    |   movel([0.162608, -1.218447, -2.664024, -0.829918, 1.570796, 1.733404],accel_mss,speed_ms,0,blend_radius_m)
    |   movel([0.161685, -1.220294, -2.663101, -0.828994, 1.570796, 1.732481],accel_mss,speed_ms,0,blend_radius_m)
    |   movel([0.160585, -1.222184, -2.662153, -0.828052, 1.570796, 1.731381],accel_mss,speed_ms,0,blend_radius_m)
    |   movel([0.163671, -1.223075, -2.661704, -0.827609, 1.570796, 1.734467],accel_mss,speed_ms,0,blend_radius_m)
    |   movel([0.165524, -1.220284, -2.663106, -0.828999, 1.570796, 1.736320],accel_mss,speed_ms,0,blend_radius_m)
    |   speed_ms = 0.005
    |   # Splitting Linear movement in 4 (instruction 1016: MoveL 952)
    |   movel([0.165524, -1.217896, -2.661930, -0.832564, 1.570796, 1.736320],accel_mss,speed_ms,0,blend_radius_m)
    |   movel([0.165524, -1.215522, -2.660749, -0.836117, 1.570796, 1.736320],accel_mss,speed_ms,0,blend_radius_m)
    |   movel([0.165524, -1.213164, -2.659566, -0.839659, 1.570796, 1.736320],accel_mss,speed_ms,0,blend_radius_m)
    |   movel([0.165524, -1.210820, -2.658378, -0.843191, 1.570796, 1.736320],accel_mss,speed_ms,0,blend_radius_m)
    |   speed_ms = 0.040
    |   # Splitting Linear movement in 8 (instruction 1018: MoveL 953)
    |   movel([0.167766, -1.211543, -2.658021, -0.842825, 1.570796, 1.738562],accel_mss,speed_ms,0,blend_radius_m)
    |   movel([0.170001, -1.212273, -2.657659, -0.842457, 1.570796, 1.740797],accel_mss,speed_ms,0,blend_radius_m)
    |   movel([0.172230, -1.213009, -2.657294, -0.842086, 1.570796, 1.743026],accel_mss,speed_ms,0,blend_radius_m)
    |   movel([0.174452, -1.213751, -2.656925, -0.841713, 1.570796, 1.745249],accel_mss,speed_ms,0,blend_radius_m)
    |   movel([0.176668, -1.214500, -2.656552, -0.841337, 1.570796, 1.747465],accel_mss,speed_ms,0,blend_radius_m)
    |   movel([0.178878, -1.215256, -2.656175, -0.840958, 1.570796, 1.749674],accel_mss,speed_ms,0,blend_radius_m)
    |   movel([0.181081, -1.216017, -2.655795, -0.840577, 1.570796, 1.751878],accel_mss,speed_ms,0,blend_radius_m)
    |   movel([0.183278, -1.216785, -2.655410, -0.840194, 1.570796, 1.754074],accel_mss,speed_ms,0,blend_radius_m)
    |   speed_ms = 0.005
    |   # Splitting Linear movement in 4 (instruction 1020: MoveL 954)
    |   movel([0.183278, -1.219124, -2.656591, -0.836674, 1.570796, 1.754074],accel_mss,speed_ms,0,blend_radius_m)
    |   movel([0.183278, -1.221477, -2.657768, -0.833145, 1.570796, 1.754074],accel_mss,speed_ms,0,blend_radius_m)
    |   movel([0.183278, -1.223844, -2.658941, -0.829604, 1.570796, 1.754074],accel_mss,speed_ms,0,blend_radius_m)
    |   movel([0.183278, -1.226226, -2.660111, -0.826052, 1.570796, 1.754074],accel_mss,speed_ms,0,blend_radius_m)
    |   speed_ms = 0.035
    |   movel([0.185050, -1.223552, -2.661464, -0.827373, 1.570796, 1.755846],accel_mss,speed_ms,0,blend_radius_m)
    |   movel([0.186685, -1.220770, -2.662863, -0.828756, 1.570796, 1.757481],accel_mss,speed_ms,0,blend_radius_m)
    |   movel([0.188167, -1.217900, -2.664296, -0.830193, 1.570796, 1.758964],accel_mss,speed_ms,0,blend_radius_m)
    |   movel([0.189493, -1.214960, -2.665755, -0.831674, 1.570796, 1.760289],accel_mss,speed_ms,0,blend_radius_m)
    |   movel([0.190642, -1.211967, -2.667230, -0.833191, 1.570796, 1.761439],accel_mss,speed_ms,0,blend_radius_m)
    |   movel([0.191604, -1.208945, -2.668710, -0.834734, 1.570796, 1.762401],accel_mss,speed_ms,0,blend_radius_m)
    |   movel([0.192368, -1.205907, -2.670187, -0.836295, 1.570796, 1.763165],accel_mss,speed_ms,0,blend_radius_m)
    |   movel([0.192919, -1.202878, -2.671649, -0.837862, 1.570796, 1.763715],accel_mss,speed_ms,0,blend_radius_m)
    |   movel([0.193243, -1.199877, -2.673088, -0.839424, 1.570796, 1.764039],accel_mss,speed_ms,0,blend_radius_m)
    |   movel([0.193330, -1.196922, -2.674495, -0.840972, 1.570796, 1.764126],accel_mss,speed_ms,0,blend_radius_m)
    |   movel([0.193159, -1.194041, -2.675858, -0.842490, 1.570796, 1.763955],accel_mss,speed_ms,0,blend_radius_m)
    |   movel([0.192720, -1.191255, -2.677167, -0.843967, 1.570796, 1.763517],accel_mss,speed_ms,0,blend_radius_m)
    |   movel([0.192000, -1.188584, -2.678414, -0.845391, 1.570796, 1.762796],accel_mss,speed_ms,0,blend_radius_m)
    |   movel([0.190984, -1.186054, -2.679588, -0.846746, 1.570796, 1.761780],accel_mss,speed_ms,0,blend_radius_m)
    |   movel([0.189658, -1.183690, -2.680680, -0.848019, 1.570796, 1.760454],accel_mss,speed_ms,0,blend_radius_m)
    |   movel([0.188006, -1.181513, -2.681679, -0.849197, 1.570796, 1.758802],accel_mss,speed_ms,0,blend_radius_m)
    |   movel([0.186034, -1.179579, -2.682563, -0.850247, 1.570796, 1.756830],accel_mss,speed_ms,0,blend_radius_m)
    |   movel([0.183805, -1.177953, -2.683303, -0.851133, 1.570796, 1.754602],accel_mss,speed_ms,0,blend_radius_m)
    |   movel([0.181340, -1.176638, -2.683899, -0.851852, 1.570796, 1.752136],accel_mss,speed_ms,0,blend_radius_m)
    |   movel([0.178653, -1.175637, -2.684352, -0.852400, 1.570796, 1.749450],accel_mss,speed_ms,0,blend_radius_m)
    |   movel([0.175765, -1.174950, -2.684662, -0.852777, 1.570796, 1.746561],accel_mss,speed_ms,0,blend_radius_m)
    |   movel([0.172695, -1.174575, -2.684831, -0.852983, 1.570796, 1.743491],accel_mss,speed_ms,0,blend_radius_m)
    |   movel([0.169469, -1.174511, -2.684860, -0.853018, 1.570796, 1.740265],accel_mss,speed_ms,0,blend_radius_m)
    |   movel([0.166102, -1.174756, -2.684749, -0.852884, 1.570796, 1.736898],accel_mss,speed_ms,0,blend_radius_m)
    |   movel([0.162621, -1.175304, -2.684502, -0.852583, 1.570796, 1.733417],accel_mss,speed_ms,0,blend_radius_m)
    |   movel([0.159044, -1.176159, -2.684116, -0.852114, 1.570796, 1.729840],accel_mss,speed_ms,0,blend_radius_m)
    |   movel([0.155393, -1.177310, -2.683594, -0.851484, 1.570796, 1.726189],accel_mss,speed_ms,0,blend_radius_m)
    |   movel([0.151692, -1.178755, -2.682938, -0.850696, 1.570796, 1.722489],accel_mss,speed_ms,0,blend_radius_m)
    |   movel([0.147964, -1.180489, -2.682147, -0.849753, 1.570796, 1.718760],accel_mss,speed_ms,0,blend_radius_m)
    |   movel([0.144226, -1.182504, -2.681225, -0.848661, 1.570796, 1.715023],accel_mss,speed_ms,0,blend_radius_m)
    |   movel([0.140507, -1.184794, -2.680171, -0.847424, 1.570796, 1.711304],accel_mss,speed_ms,0,blend_radius_m)
    |   movel([0.136826, -1.187352, -2.678987, -0.846050, 1.570796, 1.707622],accel_mss,speed_ms,0,blend_radius_m)
    |   movel([0.133191, -1.190174, -2.677673, -0.844542, 1.570796, 1.703987],accel_mss,speed_ms,0,blend_radius_m)
    |   movel([0.129733, -1.193158, -2.676274, -0.842957, 1.570796, 1.700530],accel_mss,speed_ms,0,blend_radius_m)
    |   movel([0.126470, -1.196275, -2.674802, -0.841312, 1.570796, 1.697266],accel_mss,speed_ms,0,blend_radius_m)
    |   movel([0.123412, -1.199505, -2.673266, -0.839619, 1.570796, 1.694208],accel_mss,speed_ms,0,blend_radius_m)
    |   movel([0.120568, -1.202823, -2.671675, -0.837890, 1.570796, 1.691365],accel_mss,speed_ms,0,blend_radius_m)
    |   movel([0.117952, -1.206214, -2.670038, -0.836137, 1.570796, 1.688748],accel_mss,speed_ms,0,blend_radius_m)
    |   movel([0.115566, -1.209658, -2.668362, -0.834369, 1.570796, 1.686363],accel_mss,speed_ms,0,blend_radius_m)
    |   movel([0.113428, -1.213130, -2.666659, -0.832601, 1.570796, 1.684225],accel_mss,speed_ms,0,blend_radius_m)
    |   movel([0.111540, -1.216616, -2.664935, -0.830838, 1.570796, 1.682336],accel_mss,speed_ms,0,blend_radius_m)
    |   movel([0.109910, -1.220098, -2.663199, -0.829092, 1.570796, 1.680707],accel_mss,speed_ms,0,blend_radius_m)
    |   movel([0.108548, -1.223555, -2.661462, -0.827371, 1.570796, 1.679344],accel_mss,speed_ms,0,blend_radius_m)
    |   movel([0.107464, -1.226975, -2.659731, -0.825683, 1.570796, 1.678260],accel_mss,speed_ms,0,blend_radius_m)
    |   movel([0.106659, -1.230338, -2.658015, -0.824036, 1.570796, 1.677455],accel_mss,speed_ms,0,blend_radius_m)
    |   movel([0.106148, -1.233627, -2.656324, -0.822437, 1.570796, 1.676944],accel_mss,speed_ms,0,blend_radius_m)
    |   movel([0.105928, -1.236831, -2.654665, -0.820893, 1.570796, 1.676724],accel_mss,speed_ms,0,blend_radius_m)
    |   movel([0.106013, -1.239934, -2.653047, -0.819408, 1.570796, 1.676809],accel_mss,speed_ms,0,blend_radius_m)
    |   movel([0.106368, -1.242656, -2.651618, -0.818114, 1.570796, 1.677165],accel_mss,speed_ms,0,blend_radius_m)
    |   movel([0.106979, -1.245156, -2.650298, -0.816935, 1.570796, 1.677775],accel_mss,speed_ms,0,blend_radius_m)
    |   movel([0.107817, -1.247439, -2.649086, -0.815864, 1.570796, 1.678614],accel_mss,speed_ms,0,blend_radius_m)
    |   movel([0.108863, -1.249512, -2.647981, -0.814897, 1.570796, 1.679659],accel_mss,speed_ms,0,blend_radius_m)
    |   movel([0.110091, -1.251379, -2.646980, -0.814030, 1.570796, 1.680887],accel_mss,speed_ms,0,blend_radius_m)
    |   movel([0.111476, -1.253047, -2.646083, -0.813259, 1.570796, 1.682272],accel_mss,speed_ms,0,blend_radius_m)
    |   movel([0.112995, -1.254520, -2.645288, -0.812581, 1.570796, 1.683792],accel_mss,speed_ms,0,blend_radius_m)
    |   movel([0.114629, -1.255802, -2.644593, -0.811993, 1.570796, 1.685426],accel_mss,speed_ms,0,blend_radius_m)
    |   movel([0.116356, -1.256897, -2.643999, -0.811493, 1.570796, 1.687152],accel_mss,speed_ms,0,blend_radius_m)
    |   movel([0.118150, -1.257811, -2.643502, -0.811076, 1.570796, 1.688947],accel_mss,speed_ms,0,blend_radius_m)
    |   movel([0.119994, -1.258543, -2.643103, -0.810743, 1.570796, 1.690791],accel_mss,speed_ms,0,blend_radius_m)
    |   movel([0.121863, -1.259101, -2.642798, -0.810490, 1.570796, 1.692659],accel_mss,speed_ms,0,blend_radius_m)
    |   movel([0.123738, -1.259483, -2.642589, -0.810316, 1.570796, 1.694534],accel_mss,speed_ms,0,blend_radius_m)
    |   movel([0.125599, -1.259692, -2.642475, -0.810222, 1.570796, 1.696395],accel_mss,speed_ms,0,blend_radius_m)
    |   movel([0.127421, -1.259733, -2.642453, -0.810203, 1.570796, 1.698217],accel_mss,speed_ms,0,blend_radius_m)
    |   movel([0.129187, -1.259604, -2.642523, -0.810261, 1.570796, 1.699983],accel_mss,speed_ms,0,blend_radius_m)
    |   movel([0.130799, -1.256111, -2.644426, -0.811852, 1.570796, 1.701596],accel_mss,speed_ms,0,blend_radius_m)
    |   movel([0.127034, -1.255651, -2.644675, -0.812062, 1.570796, 1.697831],accel_mss,speed_ms,0,blend_radius_m)
    |   movel([0.123670, -1.254813, -2.645129, -0.812447, 1.570796, 1.694467],accel_mss,speed_ms,0,blend_radius_m)
    |   movel([0.120699, -1.253624, -2.645772, -0.812993, 1.570796, 1.691495],accel_mss,speed_ms,0,blend_radius_m)
    |   movel([0.118110, -1.252108, -2.646588, -0.813693, 1.570796, 1.688906],accel_mss,speed_ms,0,blend_radius_m)
    |   movel([0.115901, -1.250284, -2.647567, -0.814538, 1.570796, 1.686697],accel_mss,speed_ms,0,blend_radius_m)
    |   movel([0.114064, -1.248180, -2.648692, -0.815517, 1.570796, 1.684861],accel_mss,speed_ms,0,blend_radius_m)
    |   movel([0.112599, -1.245812, -2.649950, -0.816626, 1.570796, 1.683395],accel_mss,speed_ms,0,blend_radius_m)
    |   movel([0.111497, -1.243210, -2.651326, -0.817853, 1.570796, 1.682294],accel_mss,speed_ms,0,blend_radius_m)
    |   movel([0.110757, -1.240392, -2.652807, -0.819190, 1.570796, 1.681553],accel_mss,speed_ms,0,blend_radius_m)
    |   movel([0.110373, -1.237384, -2.654378, -0.820627, 1.570796, 1.681169],accel_mss,speed_ms,0,blend_radius_m)
    |   movel([0.110346, -1.234208, -2.656024, -0.822156, 1.570796, 1.681143],accel_mss,speed_ms,0,blend_radius_m)
    |   movel([0.110668, -1.230893, -2.657731, -0.823765, 1.570796, 1.681464],accel_mss,speed_ms,0,blend_radius_m)
    |   movel([0.111341, -1.227459, -2.659485, -0.825445, 1.570796, 1.682137],accel_mss,speed_ms,0,blend_radius_m)
    |   movel([0.112362, -1.223936, -2.661270, -0.827183, 1.570796, 1.683158],accel_mss,speed_ms,0,blend_radius_m)
    |   movel([0.113724, -1.220347, -2.663074, -0.828967, 1.570796, 1.684520],accel_mss,speed_ms,0,blend_radius_m)
    |   movel([0.115426, -1.216725, -2.664880, -0.830783, 1.570796, 1.686223],accel_mss,speed_ms,0,blend_radius_m)
    |   movel([0.117544, -1.212934, -2.666755, -0.832700, 1.570796, 1.688341],accel_mss,speed_ms,0,blend_radius_m)
    |   movel([0.119932, -1.209242, -2.668565, -0.834582, 1.570796, 1.690729],accel_mss,speed_ms,0,blend_radius_m)
    |   movel([0.122570, -1.205662, -2.670305, -0.836421, 1.570796, 1.693366],accel_mss,speed_ms,0,blend_radius_m)
    |   movel([0.125434, -1.202220, -2.671966, -0.838204, 1.570796, 1.696231],accel_mss,speed_ms,0,blend_radius_m)
    |   movel([0.128500, -1.198935, -2.673537, -0.839916, 1.570796, 1.699296],accel_mss,speed_ms,0,blend_radius_m)
    |   movel([0.131747, -1.195825, -2.675015, -0.841549, 1.570796, 1.702544],accel_mss,speed_ms,0,blend_radius_m)
    |   movel([0.135148, -1.192915, -2.676388, -0.843086, 1.570796, 1.705945],accel_mss,speed_ms,0,blend_radius_m)
    |   movel([0.138679, -1.190222, -2.677650, -0.844517, 1.570796, 1.709475],accel_mss,speed_ms,0,blend_radius_m)
    |   movel([0.142314, -1.187771, -2.678792, -0.845826, 1.570796, 1.713110],accel_mss,speed_ms,0,blend_radius_m)
    |   movel([0.146026, -1.185583, -2.679806, -0.847000, 1.570796, 1.716822],accel_mss,speed_ms,0,blend_radius_m)
    |   movel([0.149789, -1.183678, -2.680685, -0.848026, 1.570796, 1.720586],accel_mss,speed_ms,0,blend_radius_m)
    |   movel([0.153576, -1.182082, -2.681418, -0.848889, 1.570796, 1.724373],accel_mss,speed_ms,0,blend_radius_m)
    |   movel([0.157357, -1.180809, -2.682001, -0.849579, 1.570796, 1.728154],accel_mss,speed_ms,0,blend_radius_m)
    |   movel([0.161105, -1.179883, -2.682424, -0.850082, 1.570796, 1.731901],accel_mss,speed_ms,0,blend_radius_m)
    |   movel([0.164790, -1.179326, -2.682678, -0.850385, 1.570796, 1.735586],accel_mss,speed_ms,0,blend_radius_m)
    |   movel([0.168388, -1.179152, -2.682757, -0.850479, 1.570796, 1.739184],accel_mss,speed_ms,0,blend_radius_m)
    |   movel([0.171744, -1.179358, -2.682664, -0.850368, 1.570796, 1.742541],accel_mss,speed_ms,0,blend_radius_m)
    |   movel([0.174813, -1.179919, -2.682408, -0.850062, 1.570796, 1.745609],accel_mss,speed_ms,0,blend_radius_m)
    |   movel([0.177595, -1.180832, -2.681991, -0.849566, 1.570796, 1.748391],accel_mss,speed_ms,0,blend_radius_m)
    |   movel([0.180079, -1.182089, -2.681415, -0.848885, 1.570796, 1.750875],accel_mss,speed_ms,0,blend_radius_m)
    |   movel([0.182267, -1.183689, -2.680680, -0.848020, 1.570796, 1.753063],accel_mss,speed_ms,0,blend_radius_m)
    |   movel([0.184151, -1.185625, -2.679787, -0.846977, 1.570796, 1.754947],accel_mss,speed_ms,0,blend_radius_m)
    |   movel([0.185731, -1.187891, -2.678736, -0.845761, 1.570796, 1.756527],accel_mss,speed_ms,0,blend_radius_m)
    |   movel([0.187008, -1.190479, -2.677530, -0.844380, 1.570796, 1.757804],accel_mss,speed_ms,0,blend_radius_m)
    |   movel([0.188195, -1.194267, -2.675751, -0.842371, 1.570796, 1.758991],accel_mss,speed_ms,0,blend_radius_m)
    |   movel([0.188551, -1.196235, -2.674821, -0.841333, 1.570796, 1.759347],accel_mss,speed_ms,0,blend_radius_m)
    |   movel([0.188803, -1.200304, -2.672884, -0.839201, 1.570796, 1.759599],accel_mss,speed_ms,0,blend_radius_m)
    |   movel([0.188703, -1.202406, -2.671876, -0.838107, 1.570796, 1.759500],accel_mss,speed_ms,0,blend_radius_m)
    |   movel([0.188070, -1.206726, -2.669790, -0.835873, 1.570796, 1.758866],accel_mss,speed_ms,0,blend_radius_m)
    |   movel([0.187544, -1.208941, -2.668712, -0.834736, 1.570796, 1.758341],accel_mss,speed_ms,0,blend_radius_m)
    |   movel([0.186076, -1.213484, -2.666484, -0.832421, 1.570796, 1.756872],accel_mss,speed_ms,0,blend_radius_m)
    |   movel([0.185142, -1.215803, -2.665338, -0.831248, 1.570796, 1.755939],accel_mss,speed_ms,0,blend_radius_m)
    |   movel([0.182886, -1.220542, -2.662977, -0.828870, 1.570796, 1.753682],accel_mss,speed_ms,0,blend_radius_m)
    |   movel([0.180136, -1.225401, -2.660529, -0.826458, 1.570796, 1.750932],accel_mss,speed_ms,0,blend_radius_m)
    |   movel([0.183278, -1.226226, -2.660111, -0.826052, 1.570796, 1.754074],accel_mss,speed_ms,0,blend_radius_m)
    |   movel([0.185050, -1.223552, -2.661464, -0.827373, 1.570796, 1.755846],accel_mss,speed_ms,0,blend_radius_m)
    |   movel([0.185168, -1.223351, -2.661566, -0.827473, 1.570796, 1.755964],accel_mss,speed_ms,0,blend_radius_m)
    |   speed_ms = 0.005
    |   # Splitting Linear movement in 6 (instruction 1141: MoveL 1073)
    |   movel([0.185168, -1.221759, -2.660784, -0.829846, 1.570796, 1.755964],accel_mss,speed_ms,0,blend_radius_m)
    |   movel([0.185168, -1.220174, -2.660000, -0.832214, 1.570796, 1.755964],accel_mss,speed_ms,0,blend_radius_m)
    |   movel([0.185168, -1.218595, -2.659216, -0.834578, 1.570796, 1.755964],accel_mss,speed_ms,0,blend_radius_m)
    |   movel([0.185168, -1.217023, -2.658429, -0.836936, 1.570796, 1.755964],accel_mss,speed_ms,0,blend_radius_m)
    |   movel([0.185168, -1.215458, -2.657641, -0.839290, 1.570796, 1.755964],accel_mss,speed_ms,0,blend_radius_m)
    |   movel([0.185168, -1.213899, -2.656851, -0.841639, 1.570796, 1.755964],accel_mss,speed_ms,0,blend_radius_m)
    |   speed_ms = 0.040
    |   # Splitting Linear movement in 8 (instruction 1143: MoveL 1074)
    |   movel([0.184772, -1.216194, -2.655706, -0.840489, 1.570796, 1.755568],accel_mss,speed_ms,0,blend_radius_m)
    |   movel([0.184379, -1.218482, -2.654559, -0.839348, 1.570796, 1.755175],accel_mss,speed_ms,0,blend_radius_m)
    |   movel([0.183987, -1.220761, -2.653409, -0.838218, 1.570796, 1.754783],accel_mss,speed_ms,0,blend_radius_m)
    |   movel([0.183597, -1.223033, -2.652258, -0.837097, 1.570796, 1.754394],accel_mss,speed_ms,0,blend_radius_m)
    |   movel([0.183210, -1.225297, -2.651106, -0.835987, 1.570796, 1.754006],accel_mss,speed_ms,0,blend_radius_m)
    |   movel([0.182824, -1.227552, -2.649951, -0.834886, 1.570796, 1.753620],accel_mss,speed_ms,0,blend_radius_m)
    |   movel([0.182440, -1.229800, -2.648795, -0.833794, 1.570796, 1.753237],accel_mss,speed_ms,0,blend_radius_m)
    |   movel([0.182059, -1.232040, -2.647636, -0.832712, 1.570796, 1.752855],accel_mss,speed_ms,0,blend_radius_m)
    |   speed_ms = 0.005
    |   # Splitting Linear movement in 6 (instruction 1145: MoveL 1075)
    |   movel([0.182059, -1.233588, -2.648412, -0.830389, 1.570796, 1.752855],accel_mss,speed_ms,0,blend_radius_m)
    |   movel([0.182059, -1.235142, -2.649187, -0.828060, 1.570796, 1.752855],accel_mss,speed_ms,0,blend_radius_m)
    |   movel([0.182059, -1.236702, -2.649960, -0.825728, 1.570796, 1.752855],accel_mss,speed_ms,0,blend_radius_m)
    |   movel([0.182059, -1.238268, -2.650731, -0.823390, 1.570796, 1.752855],accel_mss,speed_ms,0,blend_radius_m)
    |   movel([0.182059, -1.239840, -2.651501, -0.821048, 1.570796, 1.752855],accel_mss,speed_ms,0,blend_radius_m)
    |   movel([0.182059, -1.241419, -2.652269, -0.818701, 1.570796, 1.752855],accel_mss,speed_ms,0,blend_radius_m)
    |   speed_ms = 0.035
    |   movel([0.183122, -1.243030, -2.651421, -0.817938, 1.570796, 1.753919],accel_mss,speed_ms,0,blend_radius_m)
    |   movel([0.184641, -1.244306, -2.650748, -0.817335, 1.570796, 1.755437],accel_mss,speed_ms,0,blend_radius_m)
    |   movel([0.186541, -1.245244, -2.650252, -0.816893, 1.570796, 1.757337],accel_mss,speed_ms,0,blend_radius_m)
    |   movel([0.188759, -1.245835, -2.649938, -0.816616, 1.570796, 1.759556],accel_mss,speed_ms,0,blend_radius_m)
    |   movel([0.191228, -1.246070, -2.649814, -0.816505, 1.570796, 1.762025],accel_mss,speed_ms,0,blend_radius_m)
    |   movel([0.193881, -1.245946, -2.649880, -0.816564, 1.570796, 1.764677],accel_mss,speed_ms,0,blend_radius_m)
    |   movel([0.196654, -1.245446, -2.650145, -0.816798, 1.570796, 1.767451],accel_mss,speed_ms,0,blend_radius_m)
    |   movel([0.199484, -1.244559, -2.650614, -0.817216, 1.570796, 1.770280],accel_mss,speed_ms,0,blend_radius_m)
    |   movel([0.202221, -1.243359, -2.651248, -0.817782, 1.570796, 1.773017],accel_mss,speed_ms,0,blend_radius_m)
    |   movel([0.204953, -1.241866, -2.652034, -0.818489, 1.570796, 1.775749],accel_mss,speed_ms,0,blend_radius_m)
    |   movel([0.207603, -1.240139, -2.652940, -0.819310, 1.570796, 1.778399],accel_mss,speed_ms,0,blend_radius_m)
    |   movel([0.210103, -1.238236, -2.653934, -0.820219, 1.570796, 1.780900],accel_mss,speed_ms,0,blend_radius_m)
    |   movel([0.212379, -1.236210, -2.654988, -0.821191, 1.570796, 1.783175],accel_mss,speed_ms,0,blend_radius_m)
    |   movel([0.214355, -1.234122, -2.656069, -0.822198, 1.570796, 1.785152],accel_mss,speed_ms,0,blend_radius_m)
    |   movel([0.215949, -1.232031, -2.657147, -0.823212, 1.570796, 1.786746],accel_mss,speed_ms,0,blend_radius_m)
    |   movel([0.217091, -1.229993, -2.658192, -0.824204, 1.570796, 1.787887],accel_mss,speed_ms,0,blend_radius_m)
    |   movel([0.214017, -1.229333, -2.658529, -0.824527, 1.570796, 1.784814],accel_mss,speed_ms,0,blend_radius_m)
    |   movel([0.212357, -1.231453, -2.657444, -0.823493, 1.570796, 1.783154],accel_mss,speed_ms,0,blend_radius_m)
    |   movel([0.210630, -1.233383, -2.656450, -0.822556, 1.570796, 1.781426],accel_mss,speed_ms,0,blend_radius_m)
    |   movel([0.208832, -1.235131, -2.655547, -0.821711, 1.570796, 1.779628],accel_mss,speed_ms,0,blend_radius_m)
    |   movel([0.206964, -1.236689, -2.654739, -0.820961, 1.570796, 1.777760],accel_mss,speed_ms,0,blend_radius_m)
    |   movel([0.205021, -1.238058, -2.654027, -0.820304, 1.570796, 1.775817],accel_mss,speed_ms,0,blend_radius_m)
    |   movel([0.202999, -1.239242, -2.653409, -0.819738, 1.570796, 1.773795],accel_mss,speed_ms,0,blend_radius_m)
    |   movel([0.200896, -1.240234, -2.652890, -0.819265, 1.570796, 1.771693],accel_mss,speed_ms,0,blend_radius_m)
    |   movel([0.198709, -1.241032, -2.652472, -0.818885, 1.570796, 1.769506],accel_mss,speed_ms,0,blend_radius_m)
    |   movel([0.196531, -1.241607, -2.652170, -0.818612, 1.570796, 1.767327],accel_mss,speed_ms,0,blend_radius_m)
    |   movel([0.194520, -1.241904, -2.652014, -0.818471, 1.570796, 1.765316],accel_mss,speed_ms,0,blend_radius_m)
    |   movel([0.192672, -1.241931, -2.652000, -0.818458, 1.570796, 1.763468],accel_mss,speed_ms,0,blend_radius_m)
    |   movel([0.190982, -1.241697, -2.652123, -0.818569, 1.570796, 1.761779],accel_mss,speed_ms,0,blend_radius_m)
    |   movel([0.189441, -1.241211, -2.652378, -0.818800, 1.570796, 1.760237],accel_mss,speed_ms,0,blend_radius_m)
    |   movel([0.188048, -1.240476, -2.652763, -0.819149, 1.570796, 1.758845],accel_mss,speed_ms,0,blend_radius_m)
    |   movel([0.186797, -1.239502, -2.653273, -0.819614, 1.570796, 1.757594],accel_mss,speed_ms,0,blend_radius_m)
    |   movel([0.185682, -1.238298, -2.653902, -0.820189, 1.570796, 1.756478],accel_mss,speed_ms,0,blend_radius_m)
    |   movel([0.182059, -1.241419, -2.652269, -0.818701, 1.570796, 1.752855],accel_mss,speed_ms,0,blend_radius_m)
    |   movel([0.183122, -1.243030, -2.651421, -0.817938, 1.570796, 1.753919],accel_mss,speed_ms,0,blend_radius_m)
    |   movel([0.183292, -1.243170, -2.651347, -0.817872, 1.570796, 1.754088],accel_mss,speed_ms,0,blend_radius_m)
    |   speed_ms = 0.005
    |   # Splitting Linear movement in 4 (instruction 1184: MoveL 1112)
    |   movel([0.183292, -1.240806, -2.650197, -0.821386, 1.570796, 1.754088],accel_mss,speed_ms,0,blend_radius_m)
    |   movel([0.183292, -1.238457, -2.649042, -0.824890, 1.570796, 1.754088],accel_mss,speed_ms,0,blend_radius_m)
    |   movel([0.183292, -1.236121, -2.647884, -0.828384, 1.570796, 1.754088],accel_mss,speed_ms,0,blend_radius_m)
    |   movel([0.183292, -1.233799, -2.646723, -0.831867, 1.570796, 1.754088],accel_mss,speed_ms,0,blend_radius_m)
    |   speed_ms = 0.040
    |   # Splitting Linear movement in 18 (instruction 1186: MoveL 1113)
    |   movel([0.186032, -1.232959, -2.647160, -0.832270, 1.570796, 1.756828],accel_mss,speed_ms,0,blend_radius_m)
    |   movel([0.188773, -1.232124, -2.647593, -0.832672, 1.570796, 1.759569],accel_mss,speed_ms,0,blend_radius_m)
    |   movel([0.191516, -1.231293, -2.648023, -0.833073, 1.570796, 1.762312],accel_mss,speed_ms,0,blend_radius_m)
    |   movel([0.194260, -1.230468, -2.648450, -0.833471, 1.570796, 1.765056],accel_mss,speed_ms,0,blend_radius_m)
    |   movel([0.197005, -1.229647, -2.648874, -0.833868, 1.570796, 1.767802],accel_mss,speed_ms,0,blend_radius_m)
    |   movel([0.199752, -1.228831, -2.649294, -0.834264, 1.570796, 1.770548],accel_mss,speed_ms,0,blend_radius_m)
    |   movel([0.202500, -1.228021, -2.649710, -0.834658, 1.570796, 1.773297],accel_mss,speed_ms,0,blend_radius_m)
    |   movel([0.205250, -1.227215, -2.650124, -0.835050, 1.570796, 1.776046],accel_mss,speed_ms,0,blend_radius_m)
    |   movel([0.208000, -1.226415, -2.650534, -0.835440, 1.570796, 1.778796],accel_mss,speed_ms,0,blend_radius_m)
    |   movel([0.210752, -1.225620, -2.650941, -0.835829, 1.570796, 1.781548],accel_mss,speed_ms,0,blend_radius_m)
    |   movel([0.213505, -1.224829, -2.651344, -0.836215, 1.570796, 1.784301],accel_mss,speed_ms,0,blend_radius_m)
    |   movel([0.216259, -1.224045, -2.651744, -0.836600, 1.570796, 1.787055],accel_mss,speed_ms,0,blend_radius_m)
    |   movel([0.219014, -1.223265, -2.652141, -0.836983, 1.570796, 1.789810],accel_mss,speed_ms,0,blend_radius_m)
    |   movel([0.221770, -1.222490, -2.652534, -0.837365, 1.570796, 1.792566],accel_mss,speed_ms,0,blend_radius_m)
    |   movel([0.224526, -1.221721, -2.652924, -0.837744, 1.570796, 1.795323],accel_mss,speed_ms,0,blend_radius_m)
    |   movel([0.227284, -1.220958, -2.653310, -0.838121, 1.570796, 1.798081],accel_mss,speed_ms,0,blend_radius_m)
    |   movel([0.230043, -1.220199, -2.653693, -0.838496, 1.570796, 1.800839],accel_mss,speed_ms,0,blend_radius_m)
    |   movel([0.232803, -1.219446, -2.654073, -0.838869, 1.570796, 1.803599],accel_mss,speed_ms,0,blend_radius_m)
    |   speed_ms = 0.005
    |   # Splitting Linear movement in 4 (instruction 1188: MoveL 1114)
    |   movel([0.232803, -1.221782, -2.655251, -0.835356, 1.570796, 1.803599],accel_mss,speed_ms,0,blend_radius_m)
    |   movel([0.232803, -1.224133, -2.656425, -0.831831, 1.570796, 1.803599],accel_mss,speed_ms,0,blend_radius_m)
    |   movel([0.232803, -1.226497, -2.657595, -0.828296, 1.570796, 1.803599],accel_mss,speed_ms,0,blend_radius_m)
    |   movel([0.232803, -1.228877, -2.658762, -0.824750, 1.570796, 1.803599],accel_mss,speed_ms,0,blend_radius_m)
    |   speed_ms = 0.035
    |   movel([0.230920, -1.228406, -2.659003, -0.824981, 1.570796, 1.801717],accel_mss,speed_ms,0,blend_radius_m)
    |   movel([0.230264, -1.228377, -2.659017, -0.824995, 1.570796, 1.801060],accel_mss,speed_ms,0,blend_radius_m)
    |   movel([0.229709, -1.228528, -2.658940, -0.824921, 1.570796, 1.800506],accel_mss,speed_ms,0,blend_radius_m)
    |   movel([0.229199, -1.228883, -2.658759, -0.824747, 1.570796, 1.799995],accel_mss,speed_ms,0,blend_radius_m)
    |   movel([0.228657, -1.229481, -2.658454, -0.824454, 1.570796, 1.799454],accel_mss,speed_ms,0,blend_radius_m)
    |   movel([0.225246, -1.234324, -2.655964, -0.822100, 1.570796, 1.796042],accel_mss,speed_ms,0,blend_radius_m)
    |   movel([0.223109, -1.237004, -2.654575, -0.820809, 1.570796, 1.793906],accel_mss,speed_ms,0,blend_radius_m)
    |   movel([0.220844, -1.239549, -2.653248, -0.819591, 1.570796, 1.791641],accel_mss,speed_ms,0,blend_radius_m)
    |   movel([0.218468, -1.241946, -2.651992, -0.818451, 1.570796, 1.789264],accel_mss,speed_ms,0,blend_radius_m)
    |   movel([0.215996, -1.244194, -2.650807, -0.817388, 1.570796, 1.786792],accel_mss,speed_ms,0,blend_radius_m)
    |   movel([0.213445, -1.246277, -2.649704, -0.816408, 1.570796, 1.784242],accel_mss,speed_ms,0,blend_radius_m)
    |   movel([0.210829, -1.248195, -2.648684, -0.815510, 1.570796, 1.781626],accel_mss,speed_ms,0,blend_radius_m)
    |   movel([0.208160, -1.249938, -2.647752, -0.814698, 1.570796, 1.778956],accel_mss,speed_ms,0,blend_radius_m)
    |   movel([0.205457, -1.251500, -2.646915, -0.813974, 1.570796, 1.776253],accel_mss,speed_ms,0,blend_radius_m)
    |   movel([0.202731, -1.252870, -2.646178, -0.813341, 1.570796, 1.773527],accel_mss,speed_ms,0,blend_radius_m)
    |   movel([0.200000, -1.254041, -2.645547, -0.812801, 1.570796, 1.770796],accel_mss,speed_ms,0,blend_radius_m)
    |   movel([0.197273, -1.255006, -2.645025, -0.812358, 1.570796, 1.768070],accel_mss,speed_ms,0,blend_radius_m)
    |   movel([0.194565, -1.255759, -2.644617, -0.812013, 1.570796, 1.765361],accel_mss,speed_ms,0,blend_radius_m)
    |   movel([0.191894, -1.256287, -2.644330, -0.811771, 1.570796, 1.762691],accel_mss,speed_ms,0,blend_radius_m)
    |   movel([0.189269, -1.256587, -2.644168, -0.811635, 1.570796, 1.760065],accel_mss,speed_ms,0,blend_radius_m)
    |   movel([0.186708, -1.256642, -2.644138, -0.811609, 1.570796, 1.757504],accel_mss,speed_ms,0,blend_radius_m)
    |   movel([0.183681, -1.256392, -2.644274, -0.811724, 1.570796, 1.754477],accel_mss,speed_ms,0,blend_radius_m)
    |   movel([0.180930, -1.255809, -2.644590, -0.811990, 1.570796, 1.751727],accel_mss,speed_ms,0,blend_radius_m)
    |   movel([0.178461, -1.254917, -2.645073, -0.812399, 1.570796, 1.749257],accel_mss,speed_ms,0,blend_radius_m)
    |   movel([0.176271, -1.253727, -2.645716, -0.812946, 1.570796, 1.747068],accel_mss,speed_ms,0,blend_radius_m)
    |   movel([0.174378, -1.252256, -2.646509, -0.813624, 1.570796, 1.745174],accel_mss,speed_ms,0,blend_radius_m)
    |   movel([0.172780, -1.250516, -2.647443, -0.814430, 1.570796, 1.743576],accel_mss,speed_ms,0,blend_radius_m)
    |   movel([0.171488, -1.248526, -2.648507, -0.815356, 1.570796, 1.742284],accel_mss,speed_ms,0,blend_radius_m)
    |   movel([0.170509, -1.246296, -2.649694, -0.816399, 1.570796, 1.741305],accel_mss,speed_ms,0,blend_radius_m)
    |   movel([0.169853, -1.243843, -2.650993, -0.817554, 1.570796, 1.740650],accel_mss,speed_ms,0,blend_radius_m)
    |   movel([0.169531, -1.241178, -2.652395, -0.818816, 1.570796, 1.740327],accel_mss,speed_ms,0,blend_radius_m)
    |   movel([0.169549, -1.238320, -2.653890, -0.820179, 1.570796, 1.740346],accel_mss,speed_ms,0,blend_radius_m)
    |   movel([0.169920, -1.235281, -2.655470, -0.821639, 1.570796, 1.740717],accel_mss,speed_ms,0,blend_radius_m)
    |   movel([0.170655, -1.232074, -2.657124, -0.823191, 1.570796, 1.741451],accel_mss,speed_ms,0,blend_radius_m)
    |   movel([0.171759, -1.228718, -2.658843, -0.824828, 1.570796, 1.742556],accel_mss,speed_ms,0,blend_radius_m)
    |   movel([0.173248, -1.225227, -2.660617, -0.826544, 1.570796, 1.744045],accel_mss,speed_ms,0,blend_radius_m)
    |   movel([0.175135, -1.221615, -2.662439, -0.828335, 1.570796, 1.745931],accel_mss,speed_ms,0,blend_radius_m)
    |   movel([0.175741, -1.220210, -2.663143, -0.829036, 1.570796, 1.746537],accel_mss,speed_ms,0,blend_radius_m)
    |   movel([0.175768, -1.219750, -2.663373, -0.829266, 1.570796, 1.746565],accel_mss,speed_ms,0,blend_radius_m)
    |   movel([0.175649, -1.219412, -2.663542, -0.829435, 1.570796, 1.746445],accel_mss,speed_ms,0,blend_radius_m)
    |   movel([0.175056, -1.219006, -2.663745, -0.829638, 1.570796, 1.745852],accel_mss,speed_ms,0,blend_radius_m)
    |   movel([0.173610, -1.218730, -2.663883, -0.829776, 1.570796, 1.744407],accel_mss,speed_ms,0,blend_radius_m)
    |   movel([0.173153, -1.218827, -2.663834, -0.829728, 1.570796, 1.743950],accel_mss,speed_ms,0,blend_radius_m)
    |   movel([0.172770, -1.219039, -2.663728, -0.829621, 1.570796, 1.743567],accel_mss,speed_ms,0,blend_radius_m)
    |   movel([0.172444, -1.219343, -2.663576, -0.829469, 1.570796, 1.743240],accel_mss,speed_ms,0,blend_radius_m)
    |   movel([0.171457, -1.220948, -2.662774, -0.828668, 1.570796, 1.742253],accel_mss,speed_ms,0,blend_radius_m)
    |   movel([0.170206, -1.223197, -2.661643, -0.827549, 1.570796, 1.741002],accel_mss,speed_ms,0,blend_radius_m)
    |   movel([0.168132, -1.227587, -2.659419, -0.825382, 1.570796, 1.738928],accel_mss,speed_ms,0,blend_radius_m)
    |   movel([0.167304, -1.229720, -2.658331, -0.824338, 1.570796, 1.738100],accel_mss,speed_ms,0,blend_radius_m)
    |   movel([0.166050, -1.233849, -2.656210, -0.822330, 1.570796, 1.736847],accel_mss,speed_ms,0,blend_radius_m)
    |   movel([0.165319, -1.237768, -2.654178, -0.820443, 1.570796, 1.736116],accel_mss,speed_ms,0,blend_radius_m)
    |   movel([0.165086, -1.241457, -2.652249, -0.818683, 1.570796, 1.735882],accel_mss,speed_ms,0,blend_radius_m)
    |   movel([0.165329, -1.244896, -2.650436, -0.817057, 1.570796, 1.736125],accel_mss,speed_ms,0,blend_radius_m)
    |   movel([0.166030, -1.248056, -2.648758, -0.815575, 1.570796, 1.736827],accel_mss,speed_ms,0,blend_radius_m)
    |   movel([0.167168, -1.250919, -2.647227, -0.814243, 1.570796, 1.737964],accel_mss,speed_ms,0,blend_radius_m)
    |   movel([0.168727, -1.253462, -2.645859, -0.813068, 1.570796, 1.739523],accel_mss,speed_ms,0,blend_radius_m)
    |   movel([0.170690, -1.255662, -2.644670, -0.812058, 1.570796, 1.741486],accel_mss,speed_ms,0,blend_radius_m)
    |   movel([0.173040, -1.257494, -2.643675, -0.811221, 1.570796, 1.743836],accel_mss,speed_ms,0,blend_radius_m)
    |   movel([0.175759, -1.258941, -2.642885, -0.810562, 1.570796, 1.746555],accel_mss,speed_ms,0,blend_radius_m)
    |   movel([0.178840, -1.259973, -2.642321, -0.810094, 1.570796, 1.749636],accel_mss,speed_ms,0,blend_radius_m)
    |   movel([0.180510, -1.260327, -2.642128, -0.809934, 1.570796, 1.751306],accel_mss,speed_ms,0,blend_radius_m)
    |   movel([0.184106, -1.260694, -2.641927, -0.809768, 1.570796, 1.754902],accel_mss,speed_ms,0,blend_radius_m)
    |   movel([0.186028, -1.260700, -2.641923, -0.809766, 1.570796, 1.756825],accel_mss,speed_ms,0,blend_radius_m)
    |   movel([0.190118, -1.260340, -2.642121, -0.809929, 1.570796, 1.760914],accel_mss,speed_ms,0,blend_radius_m)
    |   movel([0.191256, -1.260315, -2.642134, -0.809940, 1.570796, 1.762052],accel_mss,speed_ms,0,blend_radius_m)
    |   movel([0.191977, -1.260635, -2.641959, -0.809795, 1.570796, 1.762774],accel_mss,speed_ms,0,blend_radius_m)
    |   movel([0.192328, -1.261291, -2.641599, -0.809499, 1.570796, 1.763125],accel_mss,speed_ms,0,blend_radius_m)
    |   movel([0.192350, -1.262284, -2.641053, -0.809051, 1.570796, 1.763146],accel_mss,speed_ms,0,blend_radius_m)
    |   movel([0.192192, -1.263120, -2.640593, -0.808676, 1.570796, 1.762989],accel_mss,speed_ms,0,blend_radius_m)
    |   movel([0.191509, -1.264754, -2.639691, -0.807944, 1.570796, 1.762306],accel_mss,speed_ms,0,blend_radius_m)
    |   movel([0.190999, -1.265535, -2.639259, -0.807595, 1.570796, 1.761795],accel_mss,speed_ms,0,blend_radius_m)
    |   movel([0.189676, -1.266970, -2.638462, -0.806957, 1.570796, 1.760472],accel_mss,speed_ms,0,blend_radius_m)
    |   movel([0.188880, -1.267607, -2.638108, -0.806674, 1.570796, 1.759676],accel_mss,speed_ms,0,blend_radius_m)
    |   movel([0.187157, -1.268611, -2.637549, -0.806229, 1.570796, 1.757953],accel_mss,speed_ms,0,blend_radius_m)
    |   movel([0.186313, -1.268935, -2.637368, -0.806086, 1.570796, 1.757109],accel_mss,speed_ms,0,blend_radius_m)
    |   movel([0.184714, -1.269219, -2.637209, -0.805961, 1.570796, 1.755510],accel_mss,speed_ms,0,blend_radius_m)
    |   movel([0.184004, -1.269167, -2.637238, -0.805984, 1.570796, 1.754800],accel_mss,speed_ms,0,blend_radius_m)
    |   movel([0.183383, -1.268973, -2.637347, -0.806070, 1.570796, 1.754179],accel_mss,speed_ms,0,blend_radius_m)
    |   movel([0.182873, -1.268630, -2.637538, -0.806221, 1.570796, 1.753670],accel_mss,speed_ms,0,blend_radius_m)
    |   movel([0.182496, -1.268130, -2.637817, -0.806442, 1.570796, 1.753292],accel_mss,speed_ms,0,blend_radius_m)
    |   movel([0.182072, -1.267536, -2.638148, -0.806705, 1.570796, 1.752869],accel_mss,speed_ms,0,blend_radius_m)
    |   movel([0.181586, -1.267232, -2.638317, -0.806840, 1.570796, 1.752382],accel_mss,speed_ms,0,blend_radius_m)
    |   movel([0.181046, -1.267168, -2.638352, -0.806869, 1.570796, 1.751843],accel_mss,speed_ms,0,blend_radius_m)
    |   movel([0.180458, -1.267300, -2.638279, -0.806810, 1.570796, 1.751254],accel_mss,speed_ms,0,blend_radius_m)
    |   movel([0.179180, -1.267945, -2.637920, -0.806524, 1.570796, 1.749976],accel_mss,speed_ms,0,blend_radius_m)
    |   movel([0.177812, -1.268782, -2.637453, -0.806154, 1.570796, 1.748609],accel_mss,speed_ms,0,blend_radius_m)
    |   movel([0.178144, -1.270177, -2.636673, -0.805538, 1.570796, 1.748940],accel_mss,speed_ms,0,blend_radius_m)
    |   movel([0.178747, -1.271317, -2.636035, -0.805037, 1.570796, 1.749544],accel_mss,speed_ms,0,blend_radius_m)
    |   movel([0.179596, -1.272195, -2.635542, -0.804653, 1.570796, 1.750392],accel_mss,speed_ms,0,blend_radius_m)
    |   movel([0.180671, -1.272802, -2.635200, -0.804387, 1.570796, 1.751467],accel_mss,speed_ms,0,blend_radius_m)
    |   movel([0.181946, -1.273134, -2.635013, -0.804242, 1.570796, 1.752743],accel_mss,speed_ms,0,blend_radius_m)
    |   movel([0.183398, -1.273186, -2.634984, -0.804220, 1.570796, 1.754195],accel_mss,speed_ms,0,blend_radius_m)
    |   movel([0.185006, -1.272947, -2.635118, -0.804324, 1.570796, 1.755802],accel_mss,speed_ms,0,blend_radius_m)
    |   movel([0.186748, -1.272409, -2.635421, -0.804559, 1.570796, 1.757544],accel_mss,speed_ms,0,blend_radius_m)
    |   movel([0.188676, -1.271538, -2.635910, -0.804940, 1.570796, 1.759472],accel_mss,speed_ms,0,blend_radius_m)
    |   movel([0.190397, -1.270460, -2.636515, -0.805414, 1.570796, 1.761194],accel_mss,speed_ms,0,blend_radius_m)
    |   movel([0.191925, -1.269164, -2.637240, -0.805985, 1.570796, 1.762722],accel_mss,speed_ms,0,blend_radius_m)
    |   movel([0.193267, -1.267632, -2.638094, -0.806663, 1.570796, 1.764063],accel_mss,speed_ms,0,blend_radius_m)
    |   movel([0.194432, -1.265850, -2.639084, -0.807455, 1.570796, 1.765228],accel_mss,speed_ms,0,blend_radius_m)
    |   movel([0.195428, -1.263800, -2.640218, -0.808371, 1.570796, 1.766224],accel_mss,speed_ms,0,blend_radius_m)
    |   movel([0.196267, -1.261471, -2.641500, -0.809417, 1.570796, 1.767063],accel_mss,speed_ms,0,blend_radius_m)
    |   movel([0.196954, -1.258843, -2.642939, -0.810607, 1.570796, 1.767750],accel_mss,speed_ms,0,blend_radius_m)
    |   # Splitting Linear movement in 4 (instruction 1292: MoveL 1217)
    |   movel([0.198451, -1.258274, -2.643250, -0.810865, 1.570796, 1.769247],accel_mss,speed_ms,0,blend_radius_m)
    |   movel([0.199949, -1.257705, -2.643559, -0.811124, 1.570796, 1.770745],accel_mss,speed_ms,0,blend_radius_m)
    |   movel([0.201447, -1.257138, -2.643868, -0.811383, 1.570796, 1.772244],accel_mss,speed_ms,0,blend_radius_m)
    |   movel([0.202947, -1.256572, -2.644176, -0.811641, 1.570796, 1.773743],accel_mss,speed_ms,0,blend_radius_m)
    |   # Splitting Linear movement in 4 (instruction 1293: MoveL 1218)
    |   movel([0.203300, -1.257976, -2.643412, -0.811001, 1.570796, 1.774097],accel_mss,speed_ms,0,blend_radius_m)
    |   movel([0.203653, -1.259378, -2.642647, -0.810364, 1.570796, 1.774449],accel_mss,speed_ms,0,blend_radius_m)
    |   movel([0.204004, -1.260778, -2.641880, -0.809730, 1.570796, 1.774800],accel_mss,speed_ms,0,blend_radius_m)
    |   movel([0.204354, -1.262176, -2.641113, -0.809100, 1.570796, 1.775150],accel_mss,speed_ms,0,blend_radius_m)
    |   movel([0.204524, -1.262927, -2.640699, -0.808762, 1.570796, 1.775321],accel_mss,speed_ms,0,blend_radius_m)
    |   movel([0.204547, -1.263730, -2.640257, -0.808402, 1.570796, 1.775344],accel_mss,speed_ms,0,blend_radius_m)
    |   movel([0.204425, -1.264565, -2.639796, -0.808028, 1.570796, 1.775221],accel_mss,speed_ms,0,blend_radius_m)
    |   movel([0.204155, -1.265416, -2.639325, -0.807648, 1.570796, 1.774952],accel_mss,speed_ms,0,blend_radius_m)
    |   movel([0.203744, -1.266262, -2.638856, -0.807272, 1.570796, 1.774541],accel_mss,speed_ms,0,blend_radius_m)
    |   movel([0.203186, -1.267090, -2.638395, -0.806903, 1.570796, 1.773982],accel_mss,speed_ms,0,blend_radius_m)
    |   movel([0.202483, -1.267882, -2.637955, -0.806552, 1.570796, 1.773279],accel_mss,speed_ms,0,blend_radius_m)
    |   movel([0.201639, -1.268619, -2.637544, -0.806226, 1.570796, 1.772435],accel_mss,speed_ms,0,blend_radius_m)
    |   movel([0.200711, -1.269262, -2.637185, -0.805942, 1.570796, 1.771507],accel_mss,speed_ms,0,blend_radius_m)
    |   movel([0.199711, -1.269824, -2.636871, -0.805694, 1.570796, 1.770507],accel_mss,speed_ms,0,blend_radius_m)
    |   movel([0.198711, -1.270254, -2.636630, -0.805504, 1.570796, 1.769507],accel_mss,speed_ms,0,blend_radius_m)
    |   movel([0.197772, -1.270514, -2.636485, -0.805390, 1.570796, 1.768568],accel_mss,speed_ms,0,blend_radius_m)
    |   movel([0.197038, -1.270704, -2.636378, -0.805306, 1.570796, 1.767834],accel_mss,speed_ms,0,blend_radius_m)
    |   movel([0.196425, -1.270986, -2.636220, -0.805183, 1.570796, 1.767221],accel_mss,speed_ms,0,blend_radius_m)
    |   movel([0.195918, -1.271345, -2.636019, -0.805025, 1.570796, 1.766714],accel_mss,speed_ms,0,blend_radius_m)
    |   movel([0.195505, -1.271760, -2.635786, -0.804843, 1.570796, 1.766301],accel_mss,speed_ms,0,blend_radius_m)
    |   movel([0.194906, -1.272706, -2.635254, -0.804429, 1.570796, 1.765702],accel_mss,speed_ms,0,blend_radius_m)
    |   movel([0.194513, -1.273704, -2.634691, -0.803993, 1.570796, 1.765310],accel_mss,speed_ms,0,blend_radius_m)
    |   movel([0.194667, -1.274013, -2.634517, -0.803859, 1.570796, 1.765464],accel_mss,speed_ms,0,blend_radius_m)
    |   movel([0.195204, -1.274294, -2.634358, -0.803736, 1.570796, 1.766000],accel_mss,speed_ms,0,blend_radius_m)
    |   movel([0.195929, -1.274479, -2.634254, -0.803656, 1.570796, 1.766726],accel_mss,speed_ms,0,blend_radius_m)
    |   movel([0.196658, -1.274485, -2.634251, -0.803653, 1.570796, 1.767454],accel_mss,speed_ms,0,blend_radius_m)
    |   movel([0.198004, -1.274201, -2.634411, -0.803777, 1.570796, 1.768801],accel_mss,speed_ms,0,blend_radius_m)
    |   movel([0.199317, -1.273770, -2.634655, -0.803965, 1.570796, 1.770113],accel_mss,speed_ms,0,blend_radius_m)
    |   movel([0.200588, -1.273193, -2.634979, -0.804216, 1.570796, 1.771384],accel_mss,speed_ms,0,blend_radius_m)
    |   movel([0.201817, -1.272478, -2.635382, -0.804529, 1.570796, 1.772613],accel_mss,speed_ms,0,blend_radius_m)
    |   movel([0.202994, -1.271628, -2.635860, -0.804901, 1.570796, 1.773790],accel_mss,speed_ms,0,blend_radius_m)
    |   movel([0.204120, -1.270645, -2.636411, -0.805332, 1.570796, 1.774917],accel_mss,speed_ms,0,blend_radius_m)
    |   movel([0.205190, -1.269534, -2.637033, -0.805822, 1.570796, 1.775986],accel_mss,speed_ms,0,blend_radius_m)
    |   movel([0.206199, -1.268296, -2.637724, -0.806369, 1.570796, 1.776995],accel_mss,speed_ms,0,blend_radius_m)
    |   movel([0.207103, -1.266980, -2.638457, -0.806952, 1.570796, 1.777900],accel_mss,speed_ms,0,blend_radius_m)
    |   movel([0.207807, -1.265701, -2.639167, -0.807521, 1.570796, 1.778604],accel_mss,speed_ms,0,blend_radius_m)
    |   movel([0.208315, -1.264461, -2.639853, -0.808075, 1.570796, 1.779112],accel_mss,speed_ms,0,blend_radius_m)
    |   movel([0.208637, -1.263262, -2.640515, -0.808612, 1.570796, 1.779433],accel_mss,speed_ms,0,blend_radius_m)
    |   movel([0.208784, -1.262096, -2.641157, -0.809136, 1.570796, 1.779580],accel_mss,speed_ms,0,blend_radius_m)
    |   movel([0.208759, -1.260972, -2.641774, -0.809643, 1.570796, 1.779555],accel_mss,speed_ms,0,blend_radius_m)
    |   movel([0.208572, -1.259885, -2.642369, -0.810134, 1.570796, 1.779369],accel_mss,speed_ms,0,blend_radius_m)
    |   movel([0.207897, -1.257500, -2.643671, -0.811218, 1.570796, 1.778694],accel_mss,speed_ms,0,blend_radius_m)
    |   movel([0.207905, -1.256755, -2.644076, -0.811557, 1.570796, 1.778702],accel_mss,speed_ms,0,blend_radius_m)
    |   movel([0.208101, -1.256011, -2.644480, -0.811898, 1.570796, 1.778897],accel_mss,speed_ms,0,blend_radius_m)
    |   movel([0.208573, -1.255120, -2.644963, -0.812306, 1.570796, 1.779369],accel_mss,speed_ms,0,blend_radius_m)
    |   movel([0.209207, -1.254274, -2.645421, -0.812694, 1.570796, 1.780004],accel_mss,speed_ms,0,blend_radius_m)
    |   movel([0.209973, -1.253493, -2.645843, -0.813054, 1.570796, 1.780769],accel_mss,speed_ms,0,blend_radius_m)
    |   movel([0.210836, -1.252796, -2.646218, -0.813375, 1.570796, 1.781632],accel_mss,speed_ms,0,blend_radius_m)
    |   movel([0.211761, -1.252207, -2.646535, -0.813647, 1.570796, 1.782558],accel_mss,speed_ms,0,blend_radius_m)
    |   movel([0.212715, -1.251746, -2.646783, -0.813860, 1.570796, 1.783511],accel_mss,speed_ms,0,blend_radius_m)
    |   movel([0.213660, -1.251433, -2.646951, -0.814005, 1.570796, 1.784456],accel_mss,speed_ms,0,blend_radius_m)
    |   movel([0.214566, -1.251289, -2.647028, -0.814071, 1.570796, 1.785362],accel_mss,speed_ms,0,blend_radius_m)
    |   movel([0.215386, -1.251336, -2.647003, -0.814050, 1.570796, 1.786182],accel_mss,speed_ms,0,blend_radius_m)
    |   movel([0.216119, -1.251559, -2.646883, -0.813946, 1.570796, 1.786915],accel_mss,speed_ms,0,blend_radius_m)
    |   movel([0.216742, -1.251940, -2.646679, -0.813770, 1.570796, 1.787539],accel_mss,speed_ms,0,blend_radius_m)
    |   movel([0.217226, -1.252458, -2.646400, -0.813531, 1.570796, 1.788023],accel_mss,speed_ms,0,blend_radius_m)
    |   movel([0.217546, -1.253093, -2.646058, -0.813238, 1.570796, 1.788342],accel_mss,speed_ms,0,blend_radius_m)
    |   movel([0.217674, -1.253822, -2.645665, -0.812902, 1.570796, 1.788470],accel_mss,speed_ms,0,blend_radius_m)
    |   movel([0.217589, -1.254626, -2.645231, -0.812533, 1.570796, 1.788386],accel_mss,speed_ms,0,blend_radius_m)
    |   movel([0.216822, -1.256480, -2.644226, -0.811683, 1.570796, 1.787619],accel_mss,speed_ms,0,blend_radius_m)
    |   movel([0.216645, -1.257244, -2.643810, -0.811334, 1.570796, 1.787442],accel_mss,speed_ms,0,blend_radius_m)
    |   movel([0.216707, -1.257818, -2.643498, -0.811073, 1.570796, 1.787504],accel_mss,speed_ms,0,blend_radius_m)
    |   movel([0.216977, -1.258232, -2.643273, -0.810885, 1.570796, 1.787773],accel_mss,speed_ms,0,blend_radius_m)
    |   movel([0.218033, -1.258734, -2.642999, -0.810656, 1.570796, 1.788829],accel_mss,speed_ms,0,blend_radius_m)
    |   movel([0.219586, -1.259040, -2.642832, -0.810518, 1.570796, 1.790383],accel_mss,speed_ms,0,blend_radius_m)
    |   movel([0.220854, -1.255891, -2.644546, -0.811953, 1.570796, 1.791651],accel_mss,speed_ms,0,blend_radius_m)
    |   movel([0.221397, -1.254417, -2.645344, -0.812629, 1.570796, 1.792193],accel_mss,speed_ms,0,blend_radius_m)
    |   movel([0.221758, -1.253012, -2.646102, -0.813275, 1.570796, 1.792554],accel_mss,speed_ms,0,blend_radius_m)
    |   movel([0.221874, -1.251827, -2.646739, -0.813822, 1.570796, 1.792670],accel_mss,speed_ms,0,blend_radius_m)
    |   movel([0.221785, -1.250782, -2.647300, -0.814306, 1.570796, 1.792582],accel_mss,speed_ms,0,blend_radius_m)
    |   movel([0.221506, -1.249872, -2.647788, -0.814729, 1.570796, 1.792302],accel_mss,speed_ms,0,blend_radius_m)
    |   movel([0.221046, -1.249085, -2.648209, -0.815095, 1.570796, 1.791842],accel_mss,speed_ms,0,blend_radius_m)
    |   movel([0.220424, -1.248411, -2.648568, -0.815409, 1.570796, 1.791220],accel_mss,speed_ms,0,blend_radius_m)
    |   movel([0.219648, -1.247848, -2.648869, -0.815673, 1.570796, 1.790445],accel_mss,speed_ms,0,blend_radius_m)
    |   movel([0.217698, -1.247008, -2.649315, -0.816065, 1.570796, 1.788494],accel_mss,speed_ms,0,blend_radius_m)
    |   movel([0.222139, -1.242801, -2.651542, -0.818046, 1.570796, 1.792935],accel_mss,speed_ms,0,blend_radius_m)
    |   movel([0.224204, -1.240641, -2.652677, -0.819071, 1.570796, 1.795001],accel_mss,speed_ms,0,blend_radius_m)
    |   movel([0.226161, -1.238430, -2.653833, -0.820126, 1.570796, 1.796957],accel_mss,speed_ms,0,blend_radius_m)
    |   movel([0.228003, -1.236159, -2.655015, -0.821216, 1.570796, 1.798799],accel_mss,speed_ms,0,blend_radius_m)
    |   movel([0.229726, -1.233815, -2.656227, -0.822347, 1.570796, 1.800523],accel_mss,speed_ms,0,blend_radius_m)
    |   movel([0.231330, -1.231391, -2.657475, -0.823523, 1.570796, 1.802127],accel_mss,speed_ms,0,blend_radius_m)
    |   movel([0.232803, -1.228877, -2.658762, -0.824750, 1.570796, 1.803599],accel_mss,speed_ms,0,blend_radius_m)
    |   movel([0.230920, -1.228406, -2.659003, -0.824981, 1.570796, 1.801717],accel_mss,speed_ms,0,blend_radius_m)
    |   movel([0.230427, -1.228385, -2.659013, -0.824991, 1.570796, 1.801223],accel_mss,speed_ms,0,blend_radius_m)
    |   speed_ms = 0.005
    |   # Splitting Linear movement in 4 (instruction 1375: MoveL 1299)
    |   movel([0.230427, -1.226005, -2.657846, -0.828538, 1.570796, 1.801223],accel_mss,speed_ms,0,blend_radius_m)
    |   movel([0.230427, -1.223640, -2.656675, -0.832075, 1.570796, 1.801223],accel_mss,speed_ms,0,blend_radius_m)
    |   movel([0.230427, -1.221289, -2.655500, -0.835600, 1.570796, 1.801223],accel_mss,speed_ms,0,blend_radius_m)
    |   movel([0.230427, -1.218952, -2.654322, -0.839115, 1.570796, 1.801223],accel_mss,speed_ms,0,blend_radius_m)
    |   speed_ms = 0.040
    |   # Splitting Linear movement in 6 (instruction 1377: MoveL 1300)
    |   movel([0.233415, -1.217796, -2.654903, -0.839690, 1.570796, 1.804211],accel_mss,speed_ms,0,blend_radius_m)
    |   movel([0.236407, -1.216644, -2.655481, -0.840264, 1.570796, 1.807203],accel_mss,speed_ms,0,blend_radius_m)
    |   movel([0.239402, -1.215496, -2.656055, -0.840838, 1.570796, 1.810198],accel_mss,speed_ms,0,blend_radius_m)
    |   movel([0.242400, -1.214353, -2.656625, -0.841411, 1.570796, 1.813196],accel_mss,speed_ms,0,blend_radius_m)
    |   movel([0.245401, -1.213215, -2.657192, -0.841983, 1.570796, 1.816197],accel_mss,speed_ms,0,blend_radius_m)
    |   movel([0.248406, -1.212081, -2.657754, -0.842554, 1.570796, 1.819202],accel_mss,speed_ms,0,blend_radius_m)
    |   speed_ms = 0.005
    |   # Splitting Linear movement in 4 (instruction 1379: MoveL 1301)
    |   movel([0.248406, -1.214423, -2.658940, -0.839025, 1.570796, 1.819202],accel_mss,speed_ms,0,blend_radius_m)
    |   movel([0.248406, -1.216781, -2.660123, -0.835486, 1.570796, 1.819202],accel_mss,speed_ms,0,blend_radius_m)
    |   movel([0.248406, -1.219153, -2.661301, -0.831935, 1.570796, 1.819202],accel_mss,speed_ms,0,blend_radius_m)
    |   movel([0.248406, -1.221539, -2.662477, -0.828373, 1.570796, 1.819202],accel_mss,speed_ms,0,blend_radius_m)
    |   speed_ms = 0.035
    |   movel([0.249440, -1.221100, -2.662697, -0.828592, 1.570796, 1.820237],accel_mss,speed_ms,0,blend_radius_m)
    |   movel([0.249896, -1.220618, -2.662939, -0.828832, 1.570796, 1.820692],accel_mss,speed_ms,0,blend_radius_m)
    |   movel([0.251660, -1.219328, -2.663584, -0.829477, 1.570796, 1.822457],accel_mss,speed_ms,0,blend_radius_m)
    |   movel([0.252170, -1.218877, -2.663809, -0.829703, 1.570796, 1.822966],accel_mss,speed_ms,0,blend_radius_m)
    |   movel([0.252526, -1.218380, -2.664057, -0.829952, 1.570796, 1.823322],accel_mss,speed_ms,0,blend_radius_m)
    |   movel([0.252663, -1.217814, -2.664339, -0.830236, 1.570796, 1.823460],accel_mss,speed_ms,0,blend_radius_m)
    |   movel([0.252520, -1.217162, -2.664663, -0.830563, 1.570796, 1.823317],accel_mss,speed_ms,0,blend_radius_m)
    |   movel([0.250957, -1.212895, -2.666774, -0.832720, 1.570796, 1.821754],accel_mss,speed_ms,0,blend_radius_m)
    |   movel([0.249816, -1.208349, -2.669000, -0.835039, 1.570796, 1.820612],accel_mss,speed_ms,0,blend_radius_m)
    |   movel([0.249004, -1.203570, -2.671316, -0.837503, 1.570796, 1.819800],accel_mss,speed_ms,0,blend_radius_m)
    |   movel([0.248438, -1.198603, -2.673696, -0.840090, 1.570796, 1.819234],accel_mss,speed_ms,0,blend_radius_m)
    |   movel([0.248071, -1.196971, -2.674472, -0.840946, 1.570796, 1.818867],accel_mss,speed_ms,0,blend_radius_m)
    |   movel([0.247294, -1.195707, -2.675071, -0.841611, 1.570796, 1.818090],accel_mss,speed_ms,0,blend_radius_m)
    |   movel([0.246094, -1.194851, -2.675475, -0.842062, 1.570796, 1.816891],accel_mss,speed_ms,0,blend_radius_m)
    |   movel([0.244450, -1.194456, -2.675662, -0.842271, 1.570796, 1.815247],accel_mss,speed_ms,0,blend_radius_m)
    |   movel([0.243858, -1.194529, -2.675627, -0.842232, 1.570796, 1.814654],accel_mss,speed_ms,0,blend_radius_m)
    |   movel([0.243176, -1.194765, -2.675516, -0.842108, 1.570796, 1.813973],accel_mss,speed_ms,0,blend_radius_m)
    |   movel([0.241754, -1.195353, -2.675238, -0.841798, 1.570796, 1.812550],accel_mss,speed_ms,0,blend_radius_m)
    |   movel([0.241610, -1.197173, -2.674376, -0.840840, 1.570796, 1.812406],accel_mss,speed_ms,0,blend_radius_m)
    |   movel([0.241596, -1.198038, -2.673965, -0.840386, 1.570796, 1.812393],accel_mss,speed_ms,0,blend_radius_m)
    |   movel([0.241748, -1.198782, -2.673610, -0.839997, 1.570796, 1.812545],accel_mss,speed_ms,0,blend_radius_m)
    |   movel([0.242267, -1.199690, -2.673177, -0.839522, 1.570796, 1.813063],accel_mss,speed_ms,0,blend_radius_m)
    |   movel([0.243552, -1.201321, -2.672397, -0.838671, 1.570796, 1.814349],accel_mss,speed_ms,0,blend_radius_m)
    |   movel([0.243997, -1.202262, -2.671945, -0.838182, 1.570796, 1.814793],accel_mss,speed_ms,0,blend_radius_m)
    |   movel([0.244458, -1.205464, -2.670401, -0.836524, 1.570796, 1.815254],accel_mss,speed_ms,0,blend_radius_m)
    |   movel([0.244873, -1.208689, -2.668835, -0.834866, 1.570796, 1.815669],accel_mss,speed_ms,0,blend_radius_m)
    |   # Splitting Linear movement in 6 (instruction 1407: MoveL 1328)
    |   movel([0.245470, -1.210842, -2.667782, -0.833764, 1.570796, 1.816266],accel_mss,speed_ms,0,blend_radius_m)
    |   movel([0.246063, -1.212991, -2.666727, -0.832671, 1.570796, 1.816859],accel_mss,speed_ms,0,blend_radius_m)
    |   movel([0.246653, -1.215136, -2.665668, -0.831585, 1.570796, 1.817450],accel_mss,speed_ms,0,blend_radius_m)
    |   movel([0.247240, -1.217275, -2.664607, -0.830507, 1.570796, 1.818037],accel_mss,speed_ms,0,blend_radius_m)
    |   movel([0.247825, -1.219410, -2.663543, -0.829436, 1.570796, 1.818621],accel_mss,speed_ms,0,blend_radius_m)
    |   movel([0.248406, -1.221539, -2.662477, -0.828373, 1.570796, 1.819202],accel_mss,speed_ms,0,blend_radius_m)
    |   movel([0.249440, -1.221100, -2.662697, -0.828592, 1.570796, 1.820237],accel_mss,speed_ms,0,blend_radius_m)
    |   movel([0.249896, -1.220618, -2.662939, -0.828832, 1.570796, 1.820692],accel_mss,speed_ms,0,blend_radius_m)
    |   movel([0.251259, -1.219622, -2.663437, -0.829330, 1.570796, 1.822055],accel_mss,speed_ms,0,blend_radius_m)
    |   speed_ms = 0.005
    |   # Splitting Linear movement in 6 (instruction 1412: MoveL 1332)
    |   movel([0.251259, -1.218028, -2.662653, -0.831708, 1.570796, 1.822055],accel_mss,speed_ms,0,blend_radius_m)
    |   movel([0.251259, -1.216441, -2.661866, -0.834082, 1.570796, 1.822055],accel_mss,speed_ms,0,blend_radius_m)
    |   movel([0.251259, -1.214860, -2.661079, -0.836451, 1.570796, 1.822055],accel_mss,speed_ms,0,blend_radius_m)
    |   movel([0.251259, -1.213285, -2.660289, -0.838814, 1.570796, 1.822055],accel_mss,speed_ms,0,blend_radius_m)
    |   movel([0.251259, -1.211717, -2.659499, -0.841173, 1.570796, 1.822055],accel_mss,speed_ms,0,blend_radius_m)
    |   movel([0.251259, -1.210156, -2.658706, -0.843527, 1.570796, 1.822055],accel_mss,speed_ms,0,blend_radius_m)
    |   speed_ms = 0.040
    |   # Splitting Linear movement in 14 (instruction 1414: MoveL 1333)
    |   movel([0.250067, -1.208442, -2.659550, -0.844396, 1.570796, 1.820863],accel_mss,speed_ms,0,blend_radius_m)
    |   movel([0.248869, -1.206728, -2.660391, -0.845269, 1.570796, 1.819666],accel_mss,speed_ms,0,blend_radius_m)
    |   movel([0.247667, -1.205014, -2.661229, -0.846146, 1.570796, 1.818463],accel_mss,speed_ms,0,blend_radius_m)
    |   movel([0.246458, -1.203299, -2.662064, -0.847026, 1.570796, 1.817255],accel_mss,speed_ms,0,blend_radius_m)
    |   movel([0.245244, -1.201584, -2.662896, -0.847909, 1.570796, 1.816041],accel_mss,speed_ms,0,blend_radius_m)
    |   movel([0.244025, -1.199869, -2.663724, -0.848796, 1.570796, 1.814821],accel_mss,speed_ms,0,blend_radius_m)
    |   movel([0.242800, -1.198154, -2.664549, -0.849686, 1.570796, 1.813596],accel_mss,speed_ms,0,blend_radius_m)
    |   movel([0.241569, -1.196438, -2.665372, -0.850579, 1.570796, 1.812365],accel_mss,speed_ms,0,blend_radius_m)
    |   movel([0.240332, -1.194723, -2.666191, -0.851475, 1.570796, 1.811129],accel_mss,speed_ms,0,blend_radius_m)
    |   movel([0.239090, -1.193007, -2.667007, -0.852375, 1.570796, 1.809886],accel_mss,speed_ms,0,blend_radius_m)
    |   movel([0.237842, -1.191291, -2.667819, -0.853278, 1.570796, 1.808639],accel_mss,speed_ms,0,blend_radius_m)
    |   movel([0.236589, -1.189576, -2.668629, -0.854184, 1.570796, 1.807385],accel_mss,speed_ms,0,blend_radius_m)
    |   movel([0.235329, -1.187860, -2.669435, -0.855093, 1.570796, 1.806125],accel_mss,speed_ms,0,blend_radius_m)
    |   movel([0.234064, -1.186145, -2.670239, -0.856006, 1.570796, 1.804860],accel_mss,speed_ms,0,blend_radius_m)
    |   speed_ms = 0.005
    |   # Splitting Linear movement in 6 (instruction 1416: MoveL 1334)
    |   movel([0.234064, -1.187719, -2.671049, -0.853621, 1.570796, 1.804860],accel_mss,speed_ms,0,blend_radius_m)
    |   movel([0.234064, -1.189300, -2.671858, -0.851231, 1.570796, 1.804860],accel_mss,speed_ms,0,blend_radius_m)
    |   movel([0.234064, -1.190888, -2.672665, -0.848836, 1.570796, 1.804860],accel_mss,speed_ms,0,blend_radius_m)
    |   movel([0.234064, -1.192483, -2.673471, -0.846436, 1.570796, 1.804860],accel_mss,speed_ms,0,blend_radius_m)
    |   movel([0.234064, -1.194084, -2.674275, -0.844030, 1.570796, 1.804860],accel_mss,speed_ms,0,blend_radius_m)
    |   movel([0.234064, -1.195693, -2.675078, -0.841619, 1.570796, 1.804860],accel_mss,speed_ms,0,blend_radius_m)
    |   speed_ms = 0.035
    |   movel([0.234500, -1.190747, -2.677405, -0.844237, 1.570796, 1.805297],accel_mss,speed_ms,0,blend_radius_m)
    |   movel([0.234443, -1.189222, -2.678117, -0.845050, 1.570796, 1.805239],accel_mss,speed_ms,0,blend_radius_m)
    |   movel([0.234120, -1.188848, -2.678291, -0.845250, 1.570796, 1.804916],accel_mss,speed_ms,0,blend_radius_m)
    |   movel([0.233410, -1.188682, -2.678369, -0.845339, 1.570796, 1.804207],accel_mss,speed_ms,0,blend_radius_m)
    |   movel([0.231623, -1.188484, -2.678461, -0.845444, 1.570796, 1.802419],accel_mss,speed_ms,0,blend_radius_m)
    |   movel([0.232111, -1.187021, -2.679140, -0.846227, 1.570796, 1.802907],accel_mss,speed_ms,0,blend_radius_m)
    |   movel([0.232780, -1.185639, -2.679780, -0.846969, 1.570796, 1.803577],accel_mss,speed_ms,0,blend_radius_m)
    |   movel([0.233277, -1.185016, -2.680068, -0.847304, 1.570796, 1.804073],accel_mss,speed_ms,0,blend_radius_m)
    |   movel([0.233931, -1.184463, -2.680323, -0.847602, 1.570796, 1.804728],accel_mss,speed_ms,0,blend_radius_m)
    |   movel([0.234788, -1.183991, -2.680541, -0.847857, 1.570796, 1.805584],accel_mss,speed_ms,0,blend_radius_m)
    |   movel([0.236665, -1.183355, -2.680834, -0.848201, 1.570796, 1.807461],accel_mss,speed_ms,0,blend_radius_m)
    |   movel([0.237415, -1.182980, -2.681006, -0.848403, 1.570796, 1.808212],accel_mss,speed_ms,0,blend_radius_m)
    |   movel([0.238785, -1.181931, -2.681487, -0.848970, 1.570796, 1.809581],accel_mss,speed_ms,0,blend_radius_m)
    |   movel([0.239939, -1.180565, -2.682113, -0.849711, 1.570796, 1.810736],accel_mss,speed_ms,0,blend_radius_m)
    |   movel([0.240846, -1.178954, -2.682848, -0.850588, 1.570796, 1.811642],accel_mss,speed_ms,0,blend_radius_m)
    |   movel([0.241514, -1.177140, -2.683671, -0.851577, 1.570796, 1.812310],accel_mss,speed_ms,0,blend_radius_m)
    |   movel([0.241724, -1.175563, -2.684385, -0.852441, 1.570796, 1.812520],accel_mss,speed_ms,0,blend_radius_m)
    |   movel([0.241632, -1.174874, -2.684696, -0.852819, 1.570796, 1.812428],accel_mss,speed_ms,0,blend_radius_m)
    |   movel([0.240995, -1.173736, -2.685209, -0.853444, 1.570796, 1.811791],accel_mss,speed_ms,0,blend_radius_m)
    |   movel([0.240429, -1.173300, -2.685404, -0.853684, 1.570796, 1.811225],accel_mss,speed_ms,0,blend_radius_m)
    |   movel([0.239616, -1.172699, -2.685674, -0.854015, 1.570796, 1.810413],accel_mss,speed_ms,0,blend_radius_m)
    |   movel([0.239090, -1.172037, -2.685971, -0.854381, 1.570796, 1.809886],accel_mss,speed_ms,0,blend_radius_m)
    |   movel([0.238854, -1.171309, -2.686297, -0.854783, 1.570796, 1.809650],accel_mss,speed_ms,0,blend_radius_m)
    |   movel([0.238909, -1.170504, -2.686657, -0.855228, 1.570796, 1.809705],accel_mss,speed_ms,0,blend_radius_m)
    |   movel([0.239261, -1.169610, -2.687055, -0.855724, 1.570796, 1.810058],accel_mss,speed_ms,0,blend_radius_m)
    |   movel([0.239912, -1.168627, -2.687493, -0.856269, 1.570796, 1.810709],accel_mss,speed_ms,0,blend_radius_m)
    |   movel([0.240863, -1.167540, -2.687975, -0.856874, 1.570796, 1.811659],accel_mss,speed_ms,0,blend_radius_m)
    |   movel([0.242117, -1.166348, -2.688503, -0.857538, 1.570796, 1.812914],accel_mss,speed_ms,0,blend_radius_m)
    |   movel([0.243388, -1.165101, -2.689053, -0.858235, 1.570796, 1.814184],accel_mss,speed_ms,0,blend_radius_m)
    |   movel([0.244363, -1.163828, -2.689614, -0.858947, 1.570796, 1.815160],accel_mss,speed_ms,0,blend_radius_m)
    |   movel([0.244957, -1.162512, -2.690191, -0.859686, 1.570796, 1.815754],accel_mss,speed_ms,0,blend_radius_m)
    |   movel([0.245088, -1.161125, -2.690798, -0.860466, 1.570796, 1.815884],accel_mss,speed_ms,0,blend_radius_m)
    |   movel([0.244714, -1.160041, -2.691271, -0.861078, 1.570796, 1.815511],accel_mss,speed_ms,0,blend_radius_m)
    |   movel([0.243914, -1.159611, -2.691458, -0.861320, 1.570796, 1.814710],accel_mss,speed_ms,0,blend_radius_m)
    |   movel([0.242773, -1.159629, -2.691450, -0.861310, 1.570796, 1.813569],accel_mss,speed_ms,0,blend_radius_m)
    |   movel([0.241377, -1.159892, -2.691335, -0.861162, 1.570796, 1.812174],accel_mss,speed_ms,0,blend_radius_m)
    |   movel([0.240543, -1.159815, -2.691369, -0.861205, 1.570796, 1.811340],accel_mss,speed_ms,0,blend_radius_m)
    |   movel([0.239823, -1.159334, -2.691578, -0.861477, 1.570796, 1.810619],accel_mss,speed_ms,0,blend_radius_m)
    |   movel([0.238377, -1.158026, -2.692146, -0.862217, 1.570796, 1.809174],accel_mss,speed_ms,0,blend_radius_m)
    |   movel([0.240031, -1.156826, -2.692665, -0.862897, 1.570796, 1.810827],accel_mss,speed_ms,0,blend_radius_m)
    |   movel([0.241610, -1.155880, -2.693074, -0.863435, 1.570796, 1.812406],accel_mss,speed_ms,0,blend_radius_m)
    |   movel([0.243098, -1.155182, -2.693375, -0.863832, 1.570796, 1.813894],accel_mss,speed_ms,0,blend_radius_m)
    |   movel([0.244480, -1.154735, -2.693567, -0.864086, 1.570796, 1.815276],accel_mss,speed_ms,0,blend_radius_m)
    |   movel([0.245742, -1.154537, -2.693653, -0.864200, 1.570796, 1.816538],accel_mss,speed_ms,0,blend_radius_m)
    |   movel([0.246865, -1.154585, -2.693632, -0.864172, 1.570796, 1.817661],accel_mss,speed_ms,0,blend_radius_m)
    |   movel([0.247836, -1.154874, -2.693507, -0.864007, 1.570796, 1.818633],accel_mss,speed_ms,0,blend_radius_m)
    |   movel([0.248642, -1.155408, -2.693277, -0.863703, 1.570796, 1.819438],accel_mss,speed_ms,0,blend_radius_m)
    |   movel([0.249310, -1.156229, -2.692924, -0.863237, 1.570796, 1.820106],accel_mss,speed_ms,0,blend_radius_m)
    |   movel([0.249750, -1.157258, -2.692479, -0.862652, 1.570796, 1.820546],accel_mss,speed_ms,0,blend_radius_m)
    |   movel([0.249961, -1.158455, -2.691960, -0.861974, 1.570796, 1.820758],accel_mss,speed_ms,0,blend_radius_m)
    |   movel([0.249947, -1.159767, -2.691390, -0.861232, 1.570796, 1.820743],accel_mss,speed_ms,0,blend_radius_m)
    |   movel([0.249702, -1.161157, -2.690784, -0.860448, 1.570796, 1.820498],accel_mss,speed_ms,0,blend_radius_m)
    |   movel([0.249222, -1.162575, -2.690163, -0.859650, 1.570796, 1.820019],accel_mss,speed_ms,0,blend_radius_m)
    |   movel([0.248507, -1.163984, -2.689545, -0.858860, 1.570796, 1.819303],accel_mss,speed_ms,0,blend_radius_m)
    |   movel([0.246242, -1.167092, -2.688174, -0.857123, 1.570796, 1.817038],accel_mss,speed_ms,0,blend_radius_m)
    |   movel([0.245804, -1.167852, -2.687837, -0.856700, 1.570796, 1.816600],accel_mss,speed_ms,0,blend_radius_m)
    |   movel([0.245520, -1.168555, -2.687525, -0.856309, 1.570796, 1.816316],accel_mss,speed_ms,0,blend_radius_m)
    |   movel([0.245393, -1.169224, -2.687227, -0.855938, 1.570796, 1.816189],accel_mss,speed_ms,0,blend_radius_m)
    |   movel([0.245429, -1.169877, -2.686937, -0.855576, 1.570796, 1.816226],accel_mss,speed_ms,0,blend_radius_m)
    |   movel([0.245998, -1.171209, -2.686342, -0.854838, 1.570796, 1.816794],accel_mss,speed_ms,0,blend_radius_m)
    |   movel([0.246460, -1.172370, -2.685822, -0.854197, 1.570796, 1.817257],accel_mss,speed_ms,0,blend_radius_m)
    |   movel([0.246551, -1.173786, -2.685186, -0.853417, 1.570796, 1.817347],accel_mss,speed_ms,0,blend_radius_m)
    |   movel([0.246303, -1.175396, -2.684461, -0.852533, 1.570796, 1.817100],accel_mss,speed_ms,0,blend_radius_m)
    |   movel([0.245761, -1.177134, -2.683674, -0.851581, 1.570796, 1.816558],accel_mss,speed_ms,0,blend_radius_m)
    |   movel([0.244960, -1.178936, -2.682856, -0.850597, 1.570796, 1.815756],accel_mss,speed_ms,0,blend_radius_m)
    |   movel([0.243935, -1.180744, -2.682031, -0.849614, 1.570796, 1.814732],accel_mss,speed_ms,0,blend_radius_m)
    |   movel([0.242724, -1.182491, -2.681231, -0.848667, 1.570796, 1.813521],accel_mss,speed_ms,0,blend_radius_m)
    |   movel([0.241362, -1.184122, -2.680481, -0.847787, 1.570796, 1.812159],accel_mss,speed_ms,0,blend_radius_m)
    |   movel([0.240644, -1.185014, -2.680069, -0.847306, 1.570796, 1.811440],accel_mss,speed_ms,0,blend_radius_m)
    |   movel([0.240004, -1.186017, -2.679606, -0.846766, 1.570796, 1.810800],accel_mss,speed_ms,0,blend_radius_m)
    |   movel([0.239532, -1.187014, -2.679144, -0.846231, 1.570796, 1.810328],accel_mss,speed_ms,0,blend_radius_m)
    |   movel([0.239311, -1.187884, -2.678740, -0.845765, 1.570796, 1.810108],accel_mss,speed_ms,0,blend_radius_m)
    |   # Splitting Linear movement in 4 (instruction 1490: MoveL 1407)
    |   movel([0.239187, -1.189774, -2.677859, -0.844755, 1.570796, 1.809983],accel_mss,speed_ms,0,blend_radius_m)
    |   movel([0.239063, -1.191660, -2.676977, -0.843752, 1.570796, 1.809859],accel_mss,speed_ms,0,blend_radius_m)
    |   movel([0.238940, -1.193540, -2.676094, -0.842755, 1.570796, 1.809736],accel_mss,speed_ms,0,blend_radius_m)
    |   movel([0.238817, -1.195415, -2.675209, -0.841765, 1.570796, 1.809613],accel_mss,speed_ms,0,blend_radius_m)
    |   # Splitting Linear movement in 4 (instruction 1491: MoveL 1408)
    |   movel([0.238786, -1.197232, -2.674348, -0.840809, 1.570796, 1.809583],accel_mss,speed_ms,0,blend_radius_m)
    |   movel([0.238756, -1.199045, -2.673485, -0.839859, 1.570796, 1.809552],accel_mss,speed_ms,0,blend_radius_m)
    |   movel([0.238726, -1.200853, -2.672621, -0.838915, 1.570796, 1.809522],accel_mss,speed_ms,0,blend_radius_m)
    |   movel([0.238696, -1.202657, -2.671755, -0.837977, 1.570796, 1.809492],accel_mss,speed_ms,0,blend_radius_m)
    |   # Splitting Linear movement in 4 (instruction 1492: MoveL 1409)
    |   movel([0.238761, -1.204402, -2.670915, -0.837072, 1.570796, 1.809558],accel_mss,speed_ms,0,blend_radius_m)
    |   movel([0.238827, -1.206143, -2.670073, -0.836174, 1.570796, 1.809623],accel_mss,speed_ms,0,blend_radius_m)
    |   movel([0.238892, -1.207879, -2.669229, -0.835281, 1.570796, 1.809688],accel_mss,speed_ms,0,blend_radius_m)
    |   movel([0.238956, -1.209612, -2.668384, -0.834393, 1.570796, 1.809753],accel_mss,speed_ms,0,blend_radius_m)
    |   # Splitting Linear movement in 4 (instruction 1493: MoveL 1410)
    |   movel([0.239121, -1.211284, -2.667566, -0.833539, 1.570796, 1.809917],accel_mss,speed_ms,0,blend_radius_m)
    |   movel([0.239285, -1.212952, -2.666746, -0.832691, 1.570796, 1.810082],accel_mss,speed_ms,0,blend_radius_m)
    |   movel([0.239449, -1.214617, -2.665925, -0.831847, 1.570796, 1.810245],accel_mss,speed_ms,0,blend_radius_m)
    |   movel([0.239612, -1.216278, -2.665102, -0.831008, 1.570796, 1.810408],accel_mss,speed_ms,0,blend_radius_m)
    |   # Splitting Linear movement in 4 (instruction 1494: MoveL 1411)
    |   movel([0.239879, -1.217878, -2.664307, -0.830204, 1.570796, 1.810675],accel_mss,speed_ms,0,blend_radius_m)
    |   movel([0.240145, -1.219475, -2.663511, -0.829403, 1.570796, 1.810941],accel_mss,speed_ms,0,blend_radius_m)
    |   movel([0.240410, -1.221069, -2.662713, -0.828607, 1.570796, 1.811206],accel_mss,speed_ms,0,blend_radius_m)
    |   movel([0.240674, -1.222660, -2.661913, -0.827816, 1.570796, 1.811470],accel_mss,speed_ms,0,blend_radius_m)
    |   # Splitting Linear movement in 4 (instruction 1495: MoveL 1412)
    |   movel([0.241047, -1.224186, -2.661144, -0.827059, 1.570796, 1.811844],accel_mss,speed_ms,0,blend_radius_m)
    |   movel([0.241419, -1.225710, -2.660373, -0.826306, 1.570796, 1.812216],accel_mss,speed_ms,0,blend_radius_m)
    |   movel([0.241790, -1.227232, -2.659601, -0.825557, 1.570796, 1.812586],accel_mss,speed_ms,0,blend_radius_m)
    |   movel([0.242159, -1.228750, -2.658827, -0.824812, 1.570796, 1.812955],accel_mss,speed_ms,0,blend_radius_m)
    |   # Splitting Linear movement in 4 (instruction 1496: MoveL 1413)
    |   movel([0.242641, -1.230204, -2.658084, -0.824101, 1.570796, 1.813438],accel_mss,speed_ms,0,blend_radius_m)
    |   movel([0.243122, -1.231656, -2.657339, -0.823394, 1.570796, 1.813918],accel_mss,speed_ms,0,blend_radius_m)
    |   movel([0.243601, -1.233106, -2.656593, -0.822690, 1.570796, 1.814397],accel_mss,speed_ms,0,blend_radius_m)
    |   movel([0.244078, -1.234554, -2.655846, -0.821989, 1.570796, 1.814874],accel_mss,speed_ms,0,blend_radius_m)
    |   # Splitting Linear movement in 4 (instruction 1497: MoveL 1414)
    |   movel([0.244672, -1.235936, -2.655130, -0.821323, 1.570796, 1.815469],accel_mss,speed_ms,0,blend_radius_m)
    |   movel([0.245265, -1.237316, -2.654413, -0.820660, 1.570796, 1.816061],accel_mss,speed_ms,0,blend_radius_m)
    |   movel([0.245855, -1.238695, -2.653695, -0.819999, 1.570796, 1.816651],accel_mss,speed_ms,0,blend_radius_m)
    |   movel([0.246443, -1.240072, -2.652975, -0.819342, 1.570796, 1.817239],accel_mss,speed_ms,0,blend_radius_m)
    |   movel([0.247763, -1.242624, -2.651635, -0.818130, 1.570796, 1.818559],accel_mss,speed_ms,0,blend_radius_m)
    |   movel([0.244037, -1.245858, -2.649926, -0.816605, 1.570796, 1.814834],accel_mss,speed_ms,0,blend_radius_m)
    |   movel([0.242518, -1.243536, -2.651154, -0.817698, 1.570796, 1.813314],accel_mss,speed_ms,0,blend_radius_m)
    |   # Splitting Linear movement in 4 (instruction 1501: MoveL 1418)
    |   movel([0.242021, -1.242437, -2.651733, -0.818218, 1.570796, 1.812817],accel_mss,speed_ms,0,blend_radius_m)
    |   movel([0.241523, -1.241337, -2.652312, -0.818740, 1.570796, 1.812319],accel_mss,speed_ms,0,blend_radius_m)
    |   movel([0.241023, -1.240236, -2.652889, -0.819264, 1.570796, 1.811819],accel_mss,speed_ms,0,blend_radius_m)
    |   movel([0.240522, -1.239134, -2.653465, -0.819790, 1.570796, 1.811318],accel_mss,speed_ms,0,blend_radius_m)
    |   # Splitting Linear movement in 4 (instruction 1502: MoveL 1419)
    |   movel([0.240094, -1.237987, -2.654064, -0.820338, 1.570796, 1.810890],accel_mss,speed_ms,0,blend_radius_m)
    |   movel([0.239664, -1.236839, -2.654661, -0.820889, 1.570796, 1.810460],accel_mss,speed_ms,0,blend_radius_m)
    |   movel([0.239233, -1.235689, -2.655258, -0.821442, 1.570796, 1.810030],accel_mss,speed_ms,0,blend_radius_m)
    |   movel([0.238801, -1.234539, -2.655854, -0.821997, 1.570796, 1.809597],accel_mss,speed_ms,0,blend_radius_m)
    |   # Splitting Linear movement in 4 (instruction 1503: MoveL 1420)
    |   movel([0.238439, -1.233346, -2.656470, -0.822574, 1.570796, 1.809236],accel_mss,speed_ms,0,blend_radius_m)
    |   movel([0.238077, -1.232151, -2.657085, -0.823153, 1.570796, 1.808873],accel_mss,speed_ms,0,blend_radius_m)
    |   movel([0.237713, -1.230955, -2.657699, -0.823735, 1.570796, 1.808509],accel_mss,speed_ms,0,blend_radius_m)
    |   movel([0.237348, -1.229758, -2.658312, -0.824319, 1.570796, 1.808144],accel_mss,speed_ms,0,blend_radius_m)
    |   # Splitting Linear movement in 4 (instruction 1504: MoveL 1421)
    |   movel([0.237052, -1.228516, -2.658947, -0.824927, 1.570796, 1.807848],accel_mss,speed_ms,0,blend_radius_m)
    |   movel([0.236755, -1.227272, -2.659580, -0.825537, 1.570796, 1.807551],accel_mss,speed_ms,0,blend_radius_m)
    |   movel([0.236457, -1.226027, -2.660212, -0.826150, 1.570796, 1.807254],accel_mss,speed_ms,0,blend_radius_m)
    |   movel([0.236159, -1.224780, -2.660844, -0.826765, 1.570796, 1.806955],accel_mss,speed_ms,0,blend_radius_m)
    |   # Splitting Linear movement in 4 (instruction 1505: MoveL 1422)
    |   movel([0.235926, -1.223492, -2.661495, -0.827403, 1.570796, 1.806723],accel_mss,speed_ms,0,blend_radius_m)
    |   movel([0.235693, -1.222201, -2.662144, -0.828044, 1.570796, 1.806489],accel_mss,speed_ms,0,blend_radius_m)
    |   movel([0.235459, -1.220908, -2.662793, -0.828687, 1.570796, 1.806255],accel_mss,speed_ms,0,blend_radius_m)
    |   movel([0.235224, -1.219614, -2.663441, -0.829334, 1.570796, 1.806021],accel_mss,speed_ms,0,blend_radius_m)
    |   # Splitting Linear movement in 4 (instruction 1506: MoveL 1423)
    |   movel([0.235055, -1.218278, -2.664108, -0.830003, 1.570796, 1.805852],accel_mss,speed_ms,0,blend_radius_m)
    |   movel([0.234886, -1.216940, -2.664774, -0.830675, 1.570796, 1.805682],accel_mss,speed_ms,0,blend_radius_m)
    |   movel([0.234716, -1.215599, -2.665439, -0.831351, 1.570796, 1.805512],accel_mss,speed_ms,0,blend_radius_m)
    |   movel([0.234545, -1.214256, -2.666103, -0.832030, 1.570796, 1.805341],accel_mss,speed_ms,0,blend_radius_m)
    |   # Splitting Linear movement in 4 (instruction 1507: MoveL 1424)
    |   movel([0.234437, -1.212872, -2.666785, -0.832731, 1.570796, 1.805233],accel_mss,speed_ms,0,blend_radius_m)
    |   movel([0.234328, -1.211485, -2.667467, -0.833437, 1.570796, 1.805125],accel_mss,speed_ms,0,blend_radius_m)
    |   movel([0.234220, -1.210096, -2.668148, -0.834145, 1.570796, 1.805016],accel_mss,speed_ms,0,blend_radius_m)
    |   movel([0.234110, -1.208704, -2.668827, -0.834858, 1.570796, 1.804907],accel_mss,speed_ms,0,blend_radius_m)
    |   # Splitting Linear movement in 4 (instruction 1508: MoveL 1425)
    |   movel([0.234063, -1.206822, -2.669743, -0.835824, 1.570796, 1.804859],accel_mss,speed_ms,0,blend_radius_m)
    |   movel([0.234015, -1.204935, -2.670657, -0.836797, 1.570796, 1.804812],accel_mss,speed_ms,0,blend_radius_m)
    |   movel([0.233968, -1.203043, -2.671570, -0.837776, 1.570796, 1.804764],accel_mss,speed_ms,0,blend_radius_m)
    |   movel([0.233920, -1.201146, -2.672481, -0.838762, 1.570796, 1.804716],accel_mss,speed_ms,0,blend_radius_m)
    |   movel([0.233769, -1.200816, -2.672639, -0.838934, 1.570796, 1.804565],accel_mss,speed_ms,0,blend_radius_m)
    |   movel([0.233476, -1.200605, -2.672740, -0.839044, 1.570796, 1.804273],accel_mss,speed_ms,0,blend_radius_m)
    |   movel([0.233010, -1.200539, -2.672771, -0.839079, 1.570796, 1.803807],accel_mss,speed_ms,0,blend_radius_m)
    |   movel([0.232321, -1.200662, -2.672713, -0.839015, 1.570796, 1.803117],accel_mss,speed_ms,0,blend_radius_m)
    |   movel([0.231007, -1.201178, -2.672465, -0.838746, 1.570796, 1.801803],accel_mss,speed_ms,0,blend_radius_m)
    |   movel([0.229895, -1.201948, -2.672096, -0.838345, 1.570796, 1.800692],accel_mss,speed_ms,0,blend_radius_m)
    |   movel([0.228998, -1.202959, -2.671610, -0.837820, 1.570796, 1.799794],accel_mss,speed_ms,0,blend_radius_m)
    |   movel([0.228318, -1.204207, -2.671009, -0.837173, 1.570796, 1.799114],accel_mss,speed_ms,0,blend_radius_m)
    |   movel([0.227837, -1.205530, -2.670369, -0.836490, 1.570796, 1.798634],accel_mss,speed_ms,0,blend_radius_m)
    |   movel([0.227647, -1.206711, -2.669797, -0.835881, 1.570796, 1.798443],accel_mss,speed_ms,0,blend_radius_m)
    |   movel([0.227907, -1.207656, -2.669338, -0.835395, 1.570796, 1.798703],accel_mss,speed_ms,0,blend_radius_m)
    |   movel([0.228774, -1.208284, -2.669032, -0.835073, 1.570796, 1.799570],accel_mss,speed_ms,0,blend_radius_m)
    |   movel([0.229795, -1.208731, -2.668814, -0.834844, 1.570796, 1.800591],accel_mss,speed_ms,0,blend_radius_m)
    |   movel([0.230184, -1.209055, -2.668656, -0.834678, 1.570796, 1.800980],accel_mss,speed_ms,0,blend_radius_m)
    |   movel([0.230360, -1.209487, -2.668445, -0.834457, 1.570796, 1.801156],accel_mss,speed_ms,0,blend_radius_m)
    |   movel([0.230272, -1.210923, -2.667743, -0.833723, 1.570796, 1.801068],accel_mss,speed_ms,0,blend_radius_m)
    |   movel([0.230056, -1.211471, -2.667474, -0.833444, 1.570796, 1.800852],accel_mss,speed_ms,0,blend_radius_m)
    |   movel([0.229722, -1.211910, -2.667258, -0.833220, 1.570796, 1.800518],accel_mss,speed_ms,0,blend_radius_m)
    |   movel([0.229267, -1.212251, -2.667091, -0.833047, 1.570796, 1.800063],accel_mss,speed_ms,0,blend_radius_m)
    |   movel([0.228687, -1.212496, -2.666971, -0.832923, 1.570796, 1.799483],accel_mss,speed_ms,0,blend_radius_m)
    |   movel([0.227147, -1.212718, -2.666861, -0.832810, 1.570796, 1.797944],accel_mss,speed_ms,0,blend_radius_m)
    |   movel([0.226102, -1.212657, -2.666891, -0.832841, 1.570796, 1.796899],accel_mss,speed_ms,0,blend_radius_m)
    |   movel([0.225205, -1.212414, -2.667011, -0.832964, 1.570796, 1.796002],accel_mss,speed_ms,0,blend_radius_m)
    |   movel([0.224464, -1.211996, -2.667216, -0.833177, 1.570796, 1.795260],accel_mss,speed_ms,0,blend_radius_m)
    |   movel([0.223884, -1.211405, -2.667507, -0.833478, 1.570796, 1.794681],accel_mss,speed_ms,0,blend_radius_m)
    |   movel([0.223471, -1.210650, -2.667876, -0.833862, 1.570796, 1.794268],accel_mss,speed_ms,0,blend_radius_m)
    |   movel([0.223231, -1.209738, -2.668323, -0.834329, 1.570796, 1.794028],accel_mss,speed_ms,0,blend_radius_m)
    |   movel([0.223169, -1.208673, -2.668842, -0.834873, 1.570796, 1.793965],accel_mss,speed_ms,0,blend_radius_m)
    |   movel([0.223291, -1.207465, -2.669431, -0.835493, 1.570796, 1.794087],accel_mss,speed_ms,0,blend_radius_m)
    |   movel([0.223636, -1.205963, -2.670160, -0.836266, 1.570796, 1.794432],accel_mss,speed_ms,0,blend_radius_m)
    |   movel([0.224145, -1.204510, -2.670863, -0.837017, 1.570796, 1.794941],accel_mss,speed_ms,0,blend_radius_m)
    |   movel([0.224811, -1.203121, -2.671532, -0.837736, 1.570796, 1.795607],accel_mss,speed_ms,0,blend_radius_m)
    |   movel([0.225622, -1.201815, -2.672160, -0.838414, 1.570796, 1.796419],accel_mss,speed_ms,0,blend_radius_m)
    |   movel([0.226575, -1.200598, -2.672743, -0.839048, 1.570796, 1.797371],accel_mss,speed_ms,0,blend_radius_m)
    |   movel([0.227656, -1.199491, -2.673272, -0.839625, 1.570796, 1.798452],accel_mss,speed_ms,0,blend_radius_m)
    |   movel([0.228860, -1.198503, -2.673743, -0.840143, 1.570796, 1.799657],accel_mss,speed_ms,0,blend_radius_m)
    |   movel([0.230174, -1.197657, -2.674146, -0.840586, 1.570796, 1.800970],accel_mss,speed_ms,0,blend_radius_m)
    |   movel([0.234064, -1.195693, -2.675078, -0.841619, 1.570796, 1.804860],accel_mss,speed_ms,0,blend_radius_m)
    |   movel([0.234315, -1.192869, -2.676409, -0.843110, 1.570796, 1.805111],accel_mss,speed_ms,0,blend_radius_m)
    |   speed_ms = 0.005
    |   # Splitting Linear movement in 6 (instruction 1549: MoveL 1465)
    |   movel([0.234315, -1.191259, -2.675605, -0.845525, 1.570796, 1.805111],accel_mss,speed_ms,0,blend_radius_m)
    |   movel([0.234315, -1.189656, -2.674798, -0.847935, 1.570796, 1.805111],accel_mss,speed_ms,0,blend_radius_m)
    |   movel([0.234315, -1.188059, -2.673991, -0.850339, 1.570796, 1.805111],accel_mss,speed_ms,0,blend_radius_m)
    |   movel([0.234315, -1.186470, -2.673181, -0.852738, 1.570796, 1.805111],accel_mss,speed_ms,0,blend_radius_m)
    |   movel([0.234315, -1.184888, -2.672370, -0.855131, 1.570796, 1.805111],accel_mss,speed_ms,0,blend_radius_m)
    |   movel([0.234315, -1.183312, -2.671558, -0.857519, 1.570796, 1.805111],accel_mss,speed_ms,0,blend_radius_m)
    |   speed_ms = 0.040
    |   # Splitting Linear movement in 14 (instruction 1551: MoveL 1466)
    |   movel([0.232982, -1.181845, -2.672238, -0.858306, 1.570796, 1.803778],accel_mss,speed_ms,0,blend_radius_m)
    |   movel([0.231644, -1.180379, -2.672915, -0.859095, 1.570796, 1.802440],accel_mss,speed_ms,0,blend_radius_m)
    |   movel([0.230300, -1.178914, -2.673589, -0.859885, 1.570796, 1.801096],accel_mss,speed_ms,0,blend_radius_m)
    |   movel([0.228950, -1.177451, -2.674261, -0.860677, 1.570796, 1.799747],accel_mss,speed_ms,0,blend_radius_m)
    |   movel([0.227595, -1.175989, -2.674929, -0.861471, 1.570796, 1.798392],accel_mss,speed_ms,0,blend_radius_m)
    |   movel([0.226235, -1.174528, -2.675595, -0.862266, 1.570796, 1.797031],accel_mss,speed_ms,0,blend_radius_m)
    |   movel([0.224869, -1.173069, -2.676258, -0.863062, 1.570796, 1.795665],accel_mss,speed_ms,0,blend_radius_m)
    |   movel([0.223497, -1.171611, -2.676918, -0.863860, 1.570796, 1.794293],accel_mss,speed_ms,0,blend_radius_m)
    |   movel([0.222120, -1.170154, -2.677575, -0.864660, 1.570796, 1.792916],accel_mss,speed_ms,0,blend_radius_m)
    |   movel([0.220737, -1.168699, -2.678229, -0.865461, 1.570796, 1.791533],accel_mss,speed_ms,0,blend_radius_m)
    |   movel([0.219348, -1.167246, -2.678880, -0.866263, 1.570796, 1.790144],accel_mss,speed_ms,0,blend_radius_m)
    |   movel([0.217954, -1.165794, -2.679529, -0.867066, 1.570796, 1.788750],accel_mss,speed_ms,0,blend_radius_m)
    |   movel([0.216554, -1.164344, -2.680174, -0.867871, 1.570796, 1.787350],accel_mss,speed_ms,0,blend_radius_m)
    |   movel([0.215148, -1.162895, -2.680817, -0.868677, 1.570796, 1.785944],accel_mss,speed_ms,0,blend_radius_m)
    |   speed_ms = 0.005
    |   # Splitting Linear movement in 4 (instruction 1553: MoveL 1467)
    |   movel([0.215148, -1.165274, -2.682058, -0.865057, 1.570796, 1.785944],accel_mss,speed_ms,0,blend_radius_m)
    |   movel([0.215148, -1.167669, -2.683295, -0.861424, 1.570796, 1.785944],accel_mss,speed_ms,0,blend_radius_m)
    |   movel([0.215148, -1.170081, -2.684529, -0.857779, 1.570796, 1.785944],accel_mss,speed_ms,0,blend_radius_m)
    |   movel([0.215148, -1.172508, -2.685760, -0.854121, 1.570796, 1.785944],accel_mss,speed_ms,0,blend_radius_m)
    |   speed_ms = 0.035
    |   movel([0.215496, -1.173773, -2.685192, -0.853424, 1.570796, 1.786292],accel_mss,speed_ms,0,blend_radius_m)
    |   movel([0.215567, -1.175016, -2.684632, -0.852741, 1.570796, 1.786364],accel_mss,speed_ms,0,blend_radius_m)
    |   movel([0.215364, -1.175680, -2.684332, -0.852377, 1.570796, 1.786160],accel_mss,speed_ms,0,blend_radius_m)
    |   movel([0.214937, -1.176395, -2.684009, -0.851985, 1.570796, 1.785734],accel_mss,speed_ms,0,blend_radius_m)
    |   movel([0.214225, -1.177181, -2.683653, -0.851555, 1.570796, 1.785022],accel_mss,speed_ms,0,blend_radius_m)
    |   movel([0.213184, -1.178058, -2.683255, -0.851076, 1.570796, 1.783980],accel_mss,speed_ms,0,blend_radius_m)
    |   movel([0.212418, -1.178769, -2.682932, -0.850688, 1.570796, 1.783214],accel_mss,speed_ms,0,blend_radius_m)
    |   movel([0.211892, -1.179538, -2.682581, -0.850269, 1.570796, 1.782688],accel_mss,speed_ms,0,blend_radius_m)
    |   movel([0.211594, -1.180328, -2.682221, -0.849840, 1.570796, 1.782390],accel_mss,speed_ms,0,blend_radius_m)
    |   movel([0.211512, -1.181107, -2.681865, -0.849417, 1.570796, 1.782308],accel_mss,speed_ms,0,blend_radius_m)
    |   movel([0.211641, -1.181837, -2.681531, -0.849021, 1.570796, 1.782437],accel_mss,speed_ms,0,blend_radius_m)
    |   movel([0.211965, -1.182490, -2.681231, -0.848668, 1.570796, 1.782761],accel_mss,speed_ms,0,blend_radius_m)
    |   movel([0.212481, -1.183030, -2.680983, -0.848376, 1.570796, 1.783277],accel_mss,speed_ms,0,blend_radius_m)
    |   movel([0.213179, -1.183424, -2.680802, -0.848163, 1.570796, 1.783975],accel_mss,speed_ms,0,blend_radius_m)
    |   movel([0.216880, -1.184896, -2.680124, -0.847369, 1.570796, 1.787677],accel_mss,speed_ms,0,blend_radius_m)
    |   movel([0.218608, -1.185773, -2.679718, -0.846897, 1.570796, 1.789405],accel_mss,speed_ms,0,blend_radius_m)
    |   movel([0.220133, -1.186859, -2.679216, -0.846314, 1.570796, 1.790929],accel_mss,speed_ms,0,blend_radius_m)
    |   movel([0.221025, -1.187759, -2.678798, -0.845832, 1.570796, 1.791821],accel_mss,speed_ms,0,blend_radius_m)
    |   movel([0.222367, -1.189857, -2.677821, -0.844711, 1.570796, 1.793164],accel_mss,speed_ms,0,blend_radius_m)
    |   movel([0.222822, -1.191042, -2.677267, -0.844080, 1.570796, 1.793618],accel_mss,speed_ms,0,blend_radius_m)
    |   movel([0.223312, -1.193637, -2.676048, -0.842704, 1.570796, 1.794108],accel_mss,speed_ms,0,blend_radius_m)
    |   movel([0.223348, -1.195033, -2.675389, -0.841966, 1.570796, 1.794145],accel_mss,speed_ms,0,blend_radius_m)
    |   movel([0.223248, -1.196490, -2.674700, -0.841199, 1.570796, 1.794045],accel_mss,speed_ms,0,blend_radius_m)
    |   movel([0.222651, -1.199538, -2.673250, -0.839601, 1.570796, 1.793447],accel_mss,speed_ms,0,blend_radius_m)
    |   movel([0.221536, -1.202729, -2.671721, -0.837939, 1.570796, 1.792332],accel_mss,speed_ms,0,blend_radius_m)
    |   movel([0.219921, -1.206002, -2.670141, -0.836246, 1.570796, 1.790717],accel_mss,speed_ms,0,blend_radius_m)
    |   movel([0.217815, -1.209306, -2.668534, -0.834549, 1.570796, 1.788612],accel_mss,speed_ms,0,blend_radius_m)
    |   movel([0.217091, -1.210418, -2.667990, -0.833981, 1.570796, 1.787887],accel_mss,speed_ms,0,blend_radius_m)
    |   movel([0.216507, -1.211495, -2.667462, -0.833432, 1.570796, 1.787303],accel_mss,speed_ms,0,blend_radius_m)
    |   movel([0.215752, -1.213514, -2.666469, -0.832406, 1.570796, 1.786548],accel_mss,speed_ms,0,blend_radius_m)
    |   movel([0.215530, -1.215306, -2.665584, -0.831499, 1.570796, 1.786326],accel_mss,speed_ms,0,blend_radius_m)
    |   movel([0.215812, -1.216816, -2.664835, -0.830737, 1.570796, 1.786608],accel_mss,speed_ms,0,blend_radius_m)
    |   movel([0.216570, -1.217984, -2.664254, -0.830150, 1.570796, 1.787367],accel_mss,speed_ms,0,blend_radius_m)
    |   movel([0.217786, -1.218756, -2.663870, -0.829763, 1.570796, 1.788583],accel_mss,speed_ms,0,blend_radius_m)
    |   movel([0.219430, -1.219074, -2.663711, -0.829604, 1.570796, 1.790226],accel_mss,speed_ms,0,blend_radius_m)
    |   movel([0.220408, -1.219042, -2.663727, -0.829620, 1.570796, 1.791205],accel_mss,speed_ms,0,blend_radius_m)
    |   movel([0.222956, -1.218543, -2.663976, -0.829870, 1.570796, 1.793752],accel_mss,speed_ms,0,blend_radius_m)
    |   movel([0.224445, -1.218048, -2.664222, -0.830118, 1.570796, 1.795242],accel_mss,speed_ms,0,blend_radius_m)
    |   movel([0.225247, -1.217779, -2.664357, -0.830253, 1.570796, 1.796043],accel_mss,speed_ms,0,blend_radius_m)
    |   movel([0.225834, -1.217716, -2.664388, -0.830285, 1.570796, 1.796630],accel_mss,speed_ms,0,blend_radius_m)
    |   movel([0.226243, -1.217829, -2.664332, -0.830228, 1.570796, 1.797039],accel_mss,speed_ms,0,blend_radius_m)
    |   movel([0.226496, -1.218092, -2.664201, -0.830096, 1.570796, 1.797293],accel_mss,speed_ms,0,blend_radius_m)
    |   movel([0.226664, -1.218936, -2.663780, -0.829673, 1.570796, 1.797461],accel_mss,speed_ms,0,blend_radius_m)
    |   movel([0.226566, -1.220014, -2.663241, -0.829134, 1.570796, 1.797362],accel_mss,speed_ms,0,blend_radius_m)
    |   movel([0.226415, -1.220603, -2.662947, -0.828840, 1.570796, 1.797211],accel_mss,speed_ms,0,blend_radius_m)
    |   movel([0.226168, -1.221060, -2.662717, -0.828612, 1.570796, 1.796964],accel_mss,speed_ms,0,blend_radius_m)
    |   movel([0.225458, -1.221665, -2.662414, -0.828311, 1.570796, 1.796254],accel_mss,speed_ms,0,blend_radius_m)
    |   movel([0.224613, -1.221975, -2.662258, -0.828156, 1.570796, 1.795410],accel_mss,speed_ms,0,blend_radius_m)
    |   movel([0.219938, -1.222972, -2.661756, -0.827660, 1.570796, 1.790735],accel_mss,speed_ms,0,blend_radius_m)
    |   movel([0.218064, -1.223246, -2.661619, -0.827525, 1.570796, 1.788861],accel_mss,speed_ms,0,blend_radius_m)
    |   movel([0.216326, -1.223278, -2.661602, -0.827509, 1.570796, 1.787122],accel_mss,speed_ms,0,blend_radius_m)
    |   movel([0.215237, -1.223113, -2.661685, -0.827591, 1.570796, 1.786034],accel_mss,speed_ms,0,blend_radius_m)
    |   movel([0.214274, -1.222792, -2.661847, -0.827750, 1.570796, 1.785071],accel_mss,speed_ms,0,blend_radius_m)
    |   movel([0.213435, -1.222328, -2.662081, -0.827981, 1.570796, 1.784231],accel_mss,speed_ms,0,blend_radius_m)
    |   movel([0.212132, -1.221017, -2.662739, -0.828633, 1.570796, 1.782928],accel_mss,speed_ms,0,blend_radius_m)
    |   movel([0.211669, -1.220190, -2.663153, -0.829046, 1.570796, 1.782466],accel_mss,speed_ms,0,blend_radius_m)
    |   movel([0.211129, -1.218258, -2.664118, -0.830013, 1.570796, 1.781926],accel_mss,speed_ms,0,blend_radius_m)
    |   movel([0.211054, -1.217170, -2.664659, -0.830559, 1.570796, 1.781850],accel_mss,speed_ms,0,blend_radius_m)
    |   movel([0.211301, -1.214817, -2.665826, -0.831746, 1.570796, 1.782097],accel_mss,speed_ms,0,blend_radius_m)
    |   movel([0.211629, -1.213568, -2.666443, -0.832378, 1.570796, 1.782426],accel_mss,speed_ms,0,blend_radius_m)
    |   movel([0.212696, -1.210996, -2.667707, -0.833686, 1.570796, 1.783492],accel_mss,speed_ms,0,blend_radius_m)
    |   movel([0.213436, -1.209694, -2.668344, -0.834351, 1.570796, 1.784233],accel_mss,speed_ms,0,blend_radius_m)
    |   movel([0.215990, -1.205884, -2.670198, -0.836307, 1.570796, 1.786786],accel_mss,speed_ms,0,blend_radius_m)
    |   movel([0.217288, -1.203380, -2.671407, -0.837602, 1.570796, 1.788085],accel_mss,speed_ms,0,blend_radius_m)
    |   movel([0.218199, -1.200932, -2.672583, -0.838874, 1.570796, 1.788995],accel_mss,speed_ms,0,blend_radius_m)
    |   movel([0.218709, -1.198584, -2.673705, -0.840100, 1.570796, 1.789506],accel_mss,speed_ms,0,blend_radius_m)
    |   movel([0.218807, -1.196378, -2.674753, -0.841258, 1.570796, 1.789603],accel_mss,speed_ms,0,blend_radius_m)
    |   movel([0.218474, -1.194368, -2.675704, -0.842318, 1.570796, 1.789270],accel_mss,speed_ms,0,blend_radius_m)
    |   movel([0.217699, -1.192596, -2.676538, -0.843255, 1.570796, 1.788495],accel_mss,speed_ms,0,blend_radius_m)
    |   movel([0.216465, -1.191116, -2.677232, -0.844041, 1.570796, 1.787262],accel_mss,speed_ms,0,blend_radius_m)
    |   movel([0.215129, -1.190108, -2.677703, -0.844578, 1.570796, 1.785926],accel_mss,speed_ms,0,blend_radius_m)
    |   movel([0.213608, -1.189285, -2.678087, -0.845016, 1.570796, 1.784405],accel_mss,speed_ms,0,blend_radius_m)
    |   movel([0.209305, -1.187655, -2.678846, -0.845888, 1.570796, 1.780101],accel_mss,speed_ms,0,blend_radius_m)
    |   movel([0.208498, -1.187121, -2.679094, -0.846174, 1.570796, 1.779294],accel_mss,speed_ms,0,blend_radius_m)
    |   movel([0.207839, -1.186440, -2.679410, -0.846539, 1.570796, 1.778636],accel_mss,speed_ms,0,blend_radius_m)
    |   movel([0.207340, -1.185619, -2.679790, -0.846980, 1.570796, 1.778136],accel_mss,speed_ms,0,blend_radius_m)
    |   movel([0.207014, -1.184668, -2.680229, -0.847492, 1.570796, 1.777811],accel_mss,speed_ms,0,blend_radius_m)
    |   movel([0.206876, -1.183593, -2.680724, -0.848072, 1.570796, 1.777673],accel_mss,speed_ms,0,blend_radius_m)
    |   movel([0.206937, -1.182401, -2.681272, -0.848716, 1.570796, 1.777733],accel_mss,speed_ms,0,blend_radius_m)
    |   movel([0.207215, -1.181097, -2.681869, -0.849422, 1.570796, 1.778011],accel_mss,speed_ms,0,blend_radius_m)
    |   movel([0.207644, -1.179887, -2.682422, -0.850080, 1.570796, 1.778441],accel_mss,speed_ms,0,blend_radius_m)
    |   movel([0.208236, -1.178709, -2.682959, -0.850721, 1.570796, 1.779032],accel_mss,speed_ms,0,blend_radius_m)
    |   movel([0.208985, -1.177570, -2.683477, -0.851343, 1.570796, 1.779782],accel_mss,speed_ms,0,blend_radius_m)
    |   movel([0.209896, -1.176469, -2.683976, -0.851945, 1.570796, 1.780693],accel_mss,speed_ms,0,blend_radius_m)
    |   movel([0.210965, -1.175411, -2.684454, -0.852524, 1.570796, 1.781762],accel_mss,speed_ms,0,blend_radius_m)
    |   movel([0.212199, -1.174394, -2.684912, -0.853083, 1.570796, 1.782995],accel_mss,speed_ms,0,blend_radius_m)
    |   movel([0.213592, -1.173427, -2.685348, -0.853615, 1.570796, 1.784388],accel_mss,speed_ms,0,blend_radius_m)
    |   movel([0.215148, -1.172508, -2.685760, -0.854121, 1.570796, 1.785944],accel_mss,speed_ms,0,blend_radius_m)
    |   movel([0.215496, -1.173773, -2.685192, -0.853424, 1.570796, 1.786292],accel_mss,speed_ms,0,blend_radius_m)
    |   movel([0.215567, -1.175016, -2.684632, -0.852741, 1.570796, 1.786364],accel_mss,speed_ms,0,blend_radius_m)
    |   speed_ms = 0.005
    |   # Splitting Linear movement in 6 (instruction 1646: MoveL 1558)
    |   movel([0.215567, -1.173397, -2.683814, -0.855178, 1.570796, 1.786364],accel_mss,speed_ms,0,blend_radius_m)
    |   movel([0.215567, -1.171785, -2.682994, -0.857610, 1.570796, 1.786364],accel_mss,speed_ms,0,blend_radius_m)
    |   movel([0.215567, -1.170180, -2.682173, -0.860036, 1.570796, 1.786364],accel_mss,speed_ms,0,blend_radius_m)
    |   movel([0.215567, -1.168583, -2.681350, -0.862456, 1.570796, 1.786364],accel_mss,speed_ms,0,blend_radius_m)
    |   movel([0.215567, -1.166992, -2.680526, -0.864871, 1.570796, 1.786364],accel_mss,speed_ms,0,blend_radius_m)
    |   movel([0.215567, -1.165409, -2.679700, -0.867279, 1.570796, 1.786364],accel_mss,speed_ms,0,blend_radius_m)
    |   speed_ms = 0.040
    |   # Splitting Linear movement in 12 (instruction 1648: MoveL 1559)
    |   movel([0.217405, -1.162341, -2.681062, -0.868986, 1.570796, 1.788201],accel_mss,speed_ms,0,blend_radius_m)
    |   movel([0.219253, -1.159257, -2.682421, -0.870710, 1.570796, 1.790049],accel_mss,speed_ms,0,blend_radius_m)
    |   movel([0.221112, -1.156158, -2.683778, -0.872453, 1.570796, 1.791908],accel_mss,speed_ms,0,blend_radius_m)
    |   movel([0.222983, -1.153044, -2.685131, -0.874215, 1.570796, 1.793779],accel_mss,speed_ms,0,blend_radius_m)
    |   movel([0.224864, -1.149913, -2.686481, -0.875995, 1.570796, 1.795661],accel_mss,speed_ms,0,blend_radius_m)
    |   movel([0.226758, -1.146767, -2.687828, -0.877794, 1.570796, 1.797554],accel_mss,speed_ms,0,blend_radius_m)
    |   movel([0.228663, -1.143605, -2.689172, -0.879612, 1.570796, 1.799459],accel_mss,speed_ms,0,blend_radius_m)
    |   movel([0.230579, -1.140427, -2.690513, -0.881450, 1.570796, 1.801376],accel_mss,speed_ms,0,blend_radius_m)
    |   movel([0.232508, -1.137232, -2.691850, -0.883307, 1.570796, 1.803304],accel_mss,speed_ms,0,blend_radius_m)
    |   movel([0.234448, -1.134021, -2.693185, -0.885184, 1.570796, 1.805244],accel_mss,speed_ms,0,blend_radius_m)
    |   movel([0.236400, -1.130793, -2.694516, -0.887080, 1.570796, 1.807197],accel_mss,speed_ms,0,blend_radius_m)
    |   movel([0.238365, -1.127548, -2.695844, -0.888997, 1.570796, 1.809161],accel_mss,speed_ms,0,blend_radius_m)
    |   speed_ms = 0.005
    |   # Splitting Linear movement in 6 (instruction 1650: MoveL 1560)
    |   movel([0.238365, -1.129142, -2.696698, -0.886549, 1.570796, 1.809161],accel_mss,speed_ms,0,blend_radius_m)
    |   movel([0.238365, -1.130745, -2.697550, -0.884094, 1.570796, 1.809161],accel_mss,speed_ms,0,blend_radius_m)
    |   movel([0.238365, -1.132355, -2.698401, -0.881634, 1.570796, 1.809161],accel_mss,speed_ms,0,blend_radius_m)
    |   movel([0.238365, -1.133972, -2.699250, -0.879167, 1.570796, 1.809161],accel_mss,speed_ms,0,blend_radius_m)
    |   movel([0.238365, -1.135597, -2.700098, -0.876694, 1.570796, 1.809161],accel_mss,speed_ms,0,blend_radius_m)
    |   movel([0.238365, -1.137231, -2.700944, -0.874215, 1.570796, 1.809161],accel_mss,speed_ms,0,blend_radius_m)
    |   speed_ms = 0.035
    |   movel([0.237244, -1.139056, -2.700189, -0.873144, 1.570796, 1.808041],accel_mss,speed_ms,0,blend_radius_m)
    |   movel([0.236530, -1.140637, -2.699532, -0.872220, 1.570796, 1.807326],accel_mss,speed_ms,0,blend_radius_m)
    |   movel([0.236456, -1.141293, -2.699259, -0.871837, 1.570796, 1.807252],accel_mss,speed_ms,0,blend_radius_m)
    |   movel([0.236644, -1.141829, -2.699036, -0.871525, 1.570796, 1.807440],accel_mss,speed_ms,0,blend_radius_m)
    |   movel([0.237148, -1.142232, -2.698867, -0.871290, 1.570796, 1.807944],accel_mss,speed_ms,0,blend_radius_m)
    |   movel([0.238856, -1.142834, -2.698616, -0.870939, 1.570796, 1.809652],accel_mss,speed_ms,0,blend_radius_m)
    |   movel([0.239312, -1.143546, -2.698318, -0.870525, 1.570796, 1.810108],accel_mss,speed_ms,0,blend_radius_m)
    |   movel([0.239253, -1.144551, -2.697896, -0.869942, 1.570796, 1.810049],accel_mss,speed_ms,0,blend_radius_m)
    |   movel([0.238982, -1.145150, -2.697644, -0.869594, 1.570796, 1.809779],accel_mss,speed_ms,0,blend_radius_m)
    |   movel([0.238533, -1.145801, -2.697370, -0.869218, 1.570796, 1.809329],accel_mss,speed_ms,0,blend_radius_m)
    |   movel([0.237724, -1.146588, -2.697038, -0.868762, 1.570796, 1.808520],accel_mss,speed_ms,0,blend_radius_m)
    |   movel([0.236706, -1.147296, -2.696739, -0.868353, 1.570796, 1.807503],accel_mss,speed_ms,0,blend_radius_m)
    |   movel([0.235633, -1.147857, -2.696502, -0.868030, 1.570796, 1.806429],accel_mss,speed_ms,0,blend_radius_m)
    |   movel([0.234658, -1.148196, -2.696359, -0.867834, 1.570796, 1.805454],accel_mss,speed_ms,0,blend_radius_m)
    |   movel([0.233282, -1.148410, -2.696268, -0.867711, 1.570796, 1.804078],accel_mss,speed_ms,0,blend_radius_m)
    |   movel([0.229282, -1.148566, -2.696202, -0.867621, 1.570796, 1.800079],accel_mss,speed_ms,0,blend_radius_m)
    |   movel([0.227820, -1.148866, -2.696075, -0.867448, 1.570796, 1.798617],accel_mss,speed_ms,0,blend_radius_m)
    |   movel([0.226445, -1.149370, -2.695861, -0.867158, 1.570796, 1.797242],accel_mss,speed_ms,0,blend_radius_m)
    |   movel([0.225160, -1.150070, -2.695563, -0.866756, 1.570796, 1.795956],accel_mss,speed_ms,0,blend_radius_m)
    |   movel([0.223977, -1.150961, -2.695184, -0.866244, 1.570796, 1.794773],accel_mss,speed_ms,0,blend_radius_m)
    |   movel([0.222904, -1.152028, -2.694728, -0.865633, 1.570796, 1.793700],accel_mss,speed_ms,0,blend_radius_m)
    |   movel([0.221945, -1.153266, -2.694198, -0.864925, 1.570796, 1.792742],accel_mss,speed_ms,0,blend_radius_m)
    |   movel([0.221112, -1.154665, -2.693598, -0.864127, 1.570796, 1.791908],accel_mss,speed_ms,0,blend_radius_m)
    |   movel([0.220408, -1.156218, -2.692928, -0.863243, 1.570796, 1.791204],accel_mss,speed_ms,0,blend_radius_m)
    |   movel([0.219938, -1.157630, -2.692318, -0.862441, 1.570796, 1.790734],accel_mss,speed_ms,0,blend_radius_m)
    |   movel([0.219697, -1.158891, -2.691771, -0.861727, 1.570796, 1.790493],accel_mss,speed_ms,0,blend_radius_m)
    |   movel([0.219689, -1.160000, -2.691289, -0.861101, 1.570796, 1.790485],accel_mss,speed_ms,0,blend_radius_m)
    |   movel([0.219908, -1.160971, -2.690865, -0.860553, 1.570796, 1.790705],accel_mss,speed_ms,0,blend_radius_m)
    |   movel([0.220362, -1.161802, -2.690502, -0.860085, 1.570796, 1.791158],accel_mss,speed_ms,0,blend_radius_m)
    |   movel([0.221050, -1.162501, -2.690196, -0.859692, 1.570796, 1.791847],accel_mss,speed_ms,0,blend_radius_m)
    |   movel([0.221971, -1.163077, -2.689943, -0.859369, 1.570796, 1.792768],accel_mss,speed_ms,0,blend_radius_m)
    |   movel([0.223127, -1.163532, -2.689744, -0.859113, 1.570796, 1.793923],accel_mss,speed_ms,0,blend_radius_m)
    |   movel([0.224501, -1.164087, -2.689500, -0.858802, 1.570796, 1.795298],accel_mss,speed_ms,0,blend_radius_m)
    |   movel([0.225596, -1.164803, -2.689184, -0.858401, 1.570796, 1.796392],accel_mss,speed_ms,0,blend_radius_m)
    |   movel([0.226416, -1.165684, -2.688796, -0.857909, 1.570796, 1.797212],accel_mss,speed_ms,0,blend_radius_m)
    |   movel([0.226961, -1.166734, -2.688332, -0.857323, 1.570796, 1.797757],accel_mss,speed_ms,0,blend_radius_m)
